// TIA Portal project "Hot Water Generation V.2 (29.01.2024)" (V15.1)

(* hardware
DEVICE "S7-1200 station_1"  S7-1200 Station
   slot 0: "Rack_0"  S7-1200 Rack  Rack  V1.0
   slot 1: "PLC_1"  CPU 1214C DC/DC/DC  6ES7 214-1AG40-0XB0  V4.2
   slot 2: "AI 4x16BIT_1"  SM 1231 AI4 x HF  6ES7 231-5ND32-0XB0  V2.0
   slot 3: "AI 4x16BIT_2"  SM 1231 AI4 x HF  6ES7 231-5ND32-0XB0  V2.0
DEVICE "HMI_1"  TP700 Comfort
   slot 0: "HMI_1"  TP700 Comfort  6AV2 124-0GC01-0AX0  15.1.0.0
   slot 1: "HMI_RT_1"  TP700 Comfort  6AV2 124-0GC01-0AX0  15.1.0.0
   slot 5: "HMI_1.IE_CP_1"  PROFINET Interface  15.0.1.0
      slot 1: "PROFINET Interface_1"  PROFINET Interface
         slot 1: "Port_1"  Port
         slot 2: "Port_2"  Port
   slot 7: "HMI_1.MPI/DP_CP_1"  MPI/DP Interface  15.0.1.0
*)

// ===== PLC "PLC_1"  CPU 1214C DC/DC/DC =====

VAR_GLOBAL   // PLC tag table "Default tag table"
   "steam_preassure_sensor_pin" AT %IW96 : Int;
   "preheating_pressure_sensor_pin" AT %IW98 : Int;
   "distribution_pressure_pin" AT %IW100 : Int;
   "preheating_temperature_input_pin" AT %IW102 : Int;
   "distribution_temperature_input_pin" AT %IW112 : Int;
   "preheating_upper_level_sensor" AT %I0.0 : Bool;
   "preheating_lower_level_sensor" AT %I0.1 : Bool;
   "distribution_upper_level_sensor" AT %I0.2 : Bool;
   "distribution_lower_level_sensor" AT %I0.3 : Bool;
   "heaters" AT %Q0.0 : Bool;
   "washing_out" AT %Q0.1 : Bool;
   "washing_in" AT %Q0.2 : Bool;
   "washing_pump" AT %Q0.3 : Bool;
   "steam_valve" AT %Q0.4 : Bool;
   "preheating_tank_comp_air_bubbling_valve" AT %Q0.5 : Bool;
   "soft_water_inlet_valve" AT %Q0.6 : Bool;
   "hot_water_transfer_valve" AT %Q0.7 : Bool;
   "distribution_tank_comp_air_bubbling_valve" AT %Q1.0 : Bool;
   "distribution_valve" AT %Q1.1 : Bool;
   "preheating_vent" AT %Q8.0 : Bool;
   "distribution_vent" AT %Q8.1 : Bool;
   "System_Byte" AT %MB1 : Byte;
   "FirstScan" AT %M1.0 : Bool;
   "DiagStatusUpdate" AT %M1.1 : Bool;
   "AlwaysTRUE" AT %M1.2 : Bool;
   "AlwaysFALSE" AT %M1.3 : Bool;
   "Clock_Byte" AT %MB0 : Byte;
   "Clock_10Hz" AT %M0.0 : Bool;
   "Clock_5Hz" AT %M0.1 : Bool;
   "Clock_2.5Hz" AT %M0.2 : Bool;
   "Clock_2Hz" AT %M0.3 : Bool;
   "Clock_1.25Hz" AT %M0.4 : Bool;
   "Clock_1Hz" AT %M0.5 : Bool;
   "Clock_0.625Hz" AT %M0.6 : Bool;
   "Clock_0.5Hz" AT %M0.7 : Bool;
   "alarm" AT %MW2 : Int;
   "steam_pressure_low" AT %M2.0 : Bool;
   "preaheating_tank_pressure_low" AT %M2.2 : Bool;
   "preaheating_tank_pressure_high" AT %M2.3 : Bool;
   "preheating_temperature_low" AT %M2.4 : Bool;
   "preheating_temperature_high" AT %M2.5 : Bool;
   "steam_pressure_high" AT %M2.1 : Bool;
   "distribution_pressure_low" AT %M2.6 : Bool;
   "distribution_pressure_high" AT %M2.7 : Bool;
   "distribution_temperature_low" AT %M3.0 : Bool;
   "distribution_temperature_high" AT %M3.1 : Bool;
   "preheating_tank_empty" AT %M3.2 : Bool;
   "distribution_tank_empty" AT %M3.3 : Bool;
   "distribution_vent_switch_inverted" AT %M4.0 : Bool;
   "preheating_tank_comp_air_bubbling_valve_switch" AT %M4.1 : Bool;
END_VAR

DATA_BLOCK "sensor_inputs"   // DB1
{ S7_Optimized_Access := 'FALSE' }
VERSION : 0.1
   VAR
      preheating_steam_preassure : Real;
      preheating_tank_pressure : Real;
      distribution_tank_pressure : Real;
      preheating_temperature : Real;
      distribution_temperature : Real;
      Trend : Struct
         DT_Max_Limit : Real;
         DT_Min_Limit : Real;
         PT_Max_Limit : Real;
         PT_Min_Limit : Real;
      END_STRUCT;
   END_VAR
BEGIN
END_DATA_BLOCK

DATA_BLOCK "setpoint"   // DB3
{ S7_Optimized_Access := 'FALSE' }
VERSION : 0.1
   VAR
      distribution_temperature : Real := 70.0;
      distribution_temperature_tolerance : Real := 2.0;
      preheating_temperature : Real := 70.0;
      preheating_temperature_tolerance : Real := 5.0;
      distribution_tank_pressure : Real := 2.5;
      preheating_tank_pressure : Real := 3.0;
      preheating_steam_pressure : Real := 3.2;
      preheating_steam_pressure_tolerance : Real := 0.5;
      preaheating_tank_pressure_tolerance : Real := 0.5;
      distribution_tank_pressure_tolerance : Real := 0.5;
      is_manual_mode : Bool;
      vent_set_pressure_during_inlet : Real := 2.5;
      vent_reset_pressure_during_inlet_off : Real := 2.0;
      vent_set_critical_pressure : Real := 3.5;
      vent_reset_critical_pressure : Real := 2.8;
      critical_temperature : Real := 85.0;
   END_VAR
BEGIN
END_DATA_BLOCK

DATA_BLOCK "state"   // DB4
{ S7_Optimized_Access := 'FALSE' }
VERSION : 0.1
   VAR
      heater_pulse : Bool;
      distribution_tank_full : Bool;
      distribution_tank_empty : Bool;
      preheating_tank_full : Bool;
      preheating_tank_empty : Bool;
      stop_distribution_controller : Bool;
      stop_preheating_controller : Bool;
      steam_pulse : Bool;
      preheating_steam_pressure_high : Bool;
      preheating_tank_pressure_high : Bool;
      emergency_stop : Bool;
      preheating_temperature_in_range : Bool;
      distribution_temperature_in_range : Bool;
   END_VAR
BEGIN
END_DATA_BLOCK

DATA_BLOCK "read_sensors_DB"   // DB6
{ S7_Optimized_Access := 'TRUE' }
VERSION : 0.1
// stored: InstanceOfName read_sensors
"read_sensors"
BEGIN
END_DATA_BLOCK

DATA_BLOCK "manual"   // DB7
{ S7_Optimized_Access := 'FALSE' }
VERSION : 0.1
   VAR
      steam_valve : Bool;
      preheating_tank_comp_air_valve : Bool;
      soft_water_inlet_valve : Bool;
      hot_water_transfer_valve : Bool;
      distribution_tank_comp_air_valve : Bool;
      distribution_valve : Bool;
      heater : Bool;
      preheating_vent : Bool;
      distribution_vent : Bool;
   END_VAR
BEGIN
END_DATA_BLOCK

DATA_BLOCK "control_valves"   // DB8
{ S7_Optimized_Access := 'TRUE' }
VERSION : 0.1
// stored: InstanceOfName control_valve
"control_valve"
BEGIN
END_DATA_BLOCK

DATA_BLOCK "alarm_limit"   // DB9
{ S7_Optimized_Access := 'FALSE' }
VERSION : 0.1
   VAR
      steam_pressure_low : Real;
      steam_pressure_low_delay : Time;
      steam_pressure_high : Real;
      steam_pressure_high_delay : Time;
      preaheating_tank_pressure_low : Real;
      preaheating_tank_pressure_low_delay : Time;
      preaheating_tank_pressure_high : Real;
      preaheating_tank_pressure_high_delay : Time;
      preheating_temperature_low : Real;
      preheating_temperature_low_delay : Time;
      preheating_temperature_high : Real;
      preheating_temperature_high_delay : Time;
      distribution_pressure_low : Real;
      distribution_pressure_low_delay : Time;
      distribution_pressure_high : Real;
      distribution_pressure_high_delay : Time;
      distribution_temperature_low : Real;
      distribution_temperature_low_delay : Time;
      distribution_temperature_high : Real;
      distribution_temperature_high_delay : Time;
      preheating_tank_empty : Real;
      preheating_tank_empty_delay : Time;
      distribution_tank_empty : Real;
      distribution_tank_empty_delay : Time;
   END_VAR
BEGIN
END_DATA_BLOCK

DATA_BLOCK "alarm_management_DB"   // DB10
{ S7_Optimized_Access := 'TRUE' }
VERSION : 0.1
// stored: InstanceOfName alarm_management
"alarm_management"
BEGIN
END_DATA_BLOCK

FUNCTION_BLOCK "analog_input"   // FB1, LAD
{ S7_Optimized_Access := 'TRUE' }
VERSION : 0.1
   VAR_INPUT
      sensor_min : Real;
      sensor_max : Real;
      sensor_address : Int;
   END_VAR
   VAR_OUTPUT
      Calibrated_value : Real;
   END_VAR
   VAR
      Calibration : Real;
      Scaled_value : Real;
   END_VAR
   VAR_TEMP
      norm : Real;
   END_VAR
BEGIN

REGION Network 1
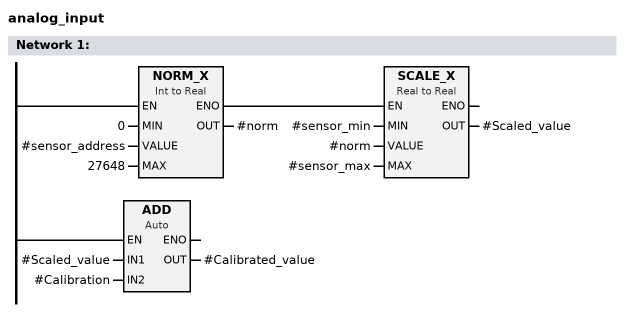
   RUNG wire#powerrail
      { S7_Templates := "[SrcType := Int, DestType := Real]" } Normalize(min := 0, value := #sensor_address, max := 27648, out => #norm)
      { S7_Templates := "[SrcType := Real, DestType := Real]" } Scale(min := #sensor_min, value := #norm, max := #sensor_max, out => #Scaled_value)
   END_RUNG
   RUNG wire#powerrail
      Add(in1 := #Scaled_value, in2 := #Calibration, out => #Calibrated_value)
   END_RUNG
   // the same network as SCL:
   #norm := NORM_X(MIN := 0, VALUE := #sensor_address, MAX := 27648);
   #Scaled_value := SCALE_X(MIN := #sensor_min, VALUE := #norm, MAX := #sensor_max);
   #Calibrated_value := #Scaled_value + #Calibration;
END_REGION
END_FUNCTION_BLOCK

FUNCTION_BLOCK "read_sensors"   // FB2, LAD
{ S7_Optimized_Access := 'TRUE' }
VERSION : 0.1
   VAR
      Steam_pressure_input : "analog_input";
      preheating_tank_pressure_input : "analog_input";
      distribution_tank_pressure_input : "analog_input";
      preheating_temperature_input : "analog_input";
      distribution_temperature_input : "analog_input";
   END_VAR
BEGIN

REGION Network 1
   // Pressure sensors
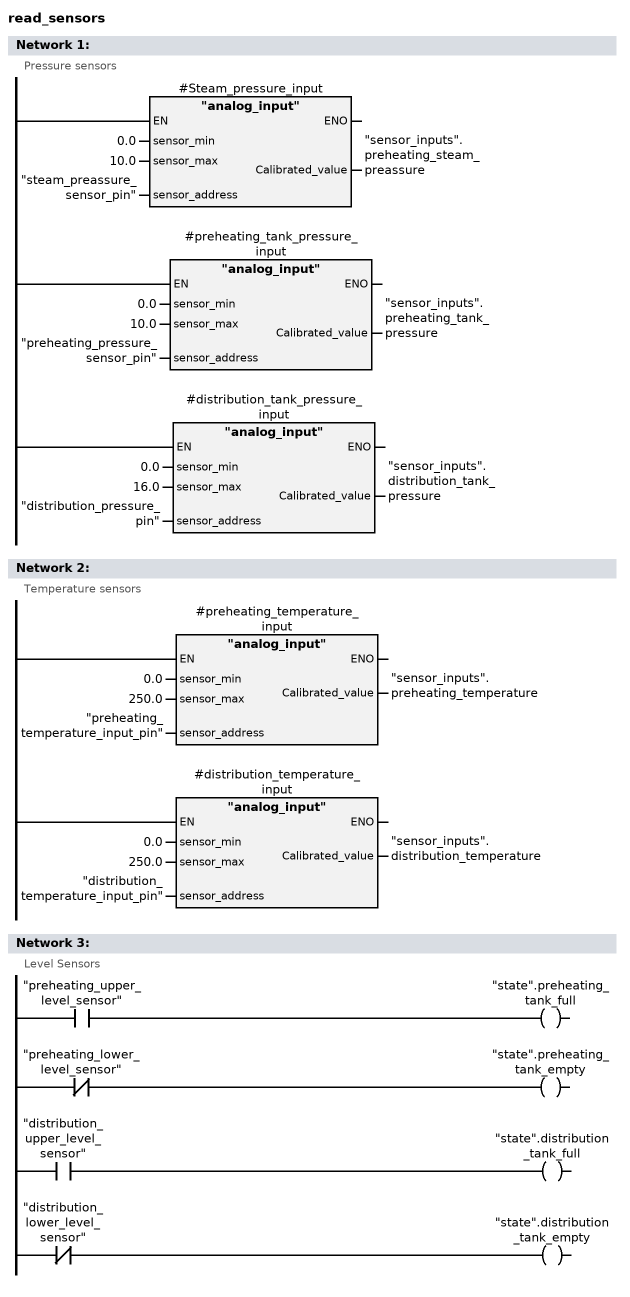
   RUNG wire#powerrail
      #Steam_pressure_input(sensor_min := 0.0, sensor_max := 10.0, sensor_address := "steam_preassure_sensor_pin", Calibrated_value => "sensor_inputs".preheating_steam_preassure)
   END_RUNG
   RUNG wire#powerrail
      #preheating_tank_pressure_input(sensor_min := 0.0, sensor_max := 10.0, sensor_address := "preheating_pressure_sensor_pin", Calibrated_value => "sensor_inputs".preheating_tank_pressure)
   END_RUNG
   RUNG wire#powerrail
      #distribution_tank_pressure_input(sensor_min := 0.0, sensor_max := 16.0, sensor_address := "distribution_pressure_pin", Calibrated_value => "sensor_inputs".distribution_tank_pressure)
   END_RUNG
   // the same network as SCL:
   #Steam_pressure_input(sensor_min := 0.0,   // "analog_input"
                         sensor_max := 10.0,
                         sensor_address := "steam_preassure_sensor_pin",
                         Calibrated_value => "sensor_inputs".preheating_steam_preassure);
   #preheating_tank_pressure_input(sensor_min := 0.0,   // "analog_input"
                           sensor_max := 10.0,
                           sensor_address := "preheating_pressure_sensor_pin",
                           Calibrated_value => "sensor_inputs".preheating_tank_pressure);
   #distribution_tank_pressure_input(sensor_min := 0.0,   // "analog_input"
                           sensor_max := 16.0,
                           sensor_address := "distribution_pressure_pin",
                           Calibrated_value => "sensor_inputs".distribution_tank_pressure);
END_REGION

REGION Network 2
   // Temperature sensors
   RUNG wire#powerrail
      #preheating_temperature_input(sensor_min := 0.0, sensor_max := 250.0, sensor_address := "preheating_temperature_input_pin", Calibrated_value => "sensor_inputs".preheating_temperature)
   END_RUNG
   RUNG wire#powerrail
      #distribution_temperature_input(sensor_min := 0.0, sensor_max := 250.0, sensor_address := "distribution_temperature_input_pin", Calibrated_value => "sensor_inputs".distribution_temperature)
   END_RUNG
   // the same network as SCL:
   #preheating_temperature_input(sensor_min := 0.0,   // "analog_input"
                           sensor_max := 250.0,
                           sensor_address := "preheating_temperature_input_pin",
                           Calibrated_value => "sensor_inputs".preheating_temperature);
   #distribution_temperature_input(sensor_min := 0.0,   // "analog_input"
                           sensor_max := 250.0,
                           sensor_address := "distribution_temperature_input_pin",
                           Calibrated_value => "sensor_inputs".distribution_temperature);
END_REGION

REGION Network 3
   // Level Sensors
   RUNG wire#powerrail
      Contact( "preheating_upper_level_sensor" )
      Coil( "state".preheating_tank_full )
   END_RUNG
   RUNG wire#powerrail
      I_Contact( "preheating_lower_level_sensor" )
      Coil( "state".preheating_tank_empty )
   END_RUNG
   RUNG wire#powerrail
      Contact( "distribution_upper_level_sensor" )
      Coil( "state".distribution_tank_full )
   END_RUNG
   RUNG wire#powerrail
      I_Contact( "distribution_lower_level_sensor" )
      Coil( "state".distribution_tank_empty )
   END_RUNG
   // the same network as SCL:
   "state".preheating_tank_full := "preheating_upper_level_sensor";
   "state".preheating_tank_empty := NOT "preheating_lower_level_sensor";
   "state".distribution_tank_full := "distribution_upper_level_sensor";
   "state".distribution_tank_empty := NOT "distribution_lower_level_sensor";
END_REGION
END_FUNCTION_BLOCK

FUNCTION_BLOCK "valve_controller_within_range"   // FB3, LAD
{ S7_Optimized_Access := 'TRUE' }
VERSION : 0.1
   VAR_INPUT
      setpoint : Real;
      current : Real;
      tolerance : Real;
      manual_switch : Bool;
   END_VAR
   VAR_OUTPUT
      output : Bool;
   END_VAR
   VAR_TEMP
      lower_trigger_point : Real;
      higher_trigger_point : Real;
   END_VAR
BEGIN

REGION Network 1
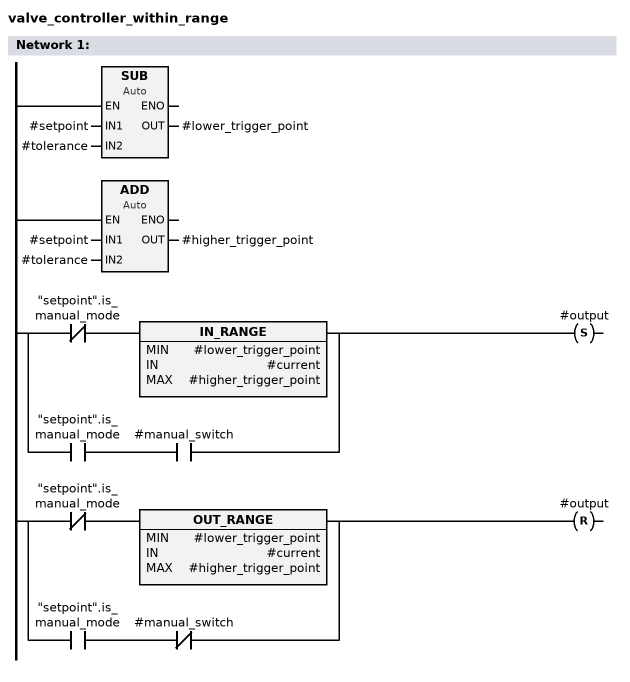
   #lower_trigger_point := #setpoint - #tolerance;
   #higher_trigger_point := #setpoint + #tolerance;
   IF (NOT "setpoint".is_manual_mode AND (#lower_trigger_point <= #current) AND (#current <= #higher_trigger_point)) OR ("setpoint".is_manual_mode AND #manual_switch) THEN
       #output := TRUE;
   END_IF;
   IF (NOT "setpoint".is_manual_mode AND ((#current < #lower_trigger_point) OR (#current > #higher_trigger_point))) OR ("setpoint".is_manual_mode AND NOT #manual_switch) THEN
       #output := FALSE;
   END_IF;
END_REGION
END_FUNCTION_BLOCK

FUNCTION_BLOCK "pressure_controller"   // FB4, LAD
{ S7_Optimized_Access := 'TRUE' }
VERSION : 0.1
   VAR
      tank_1_steam_valve_controller : "valve_controller_within_range";
   END_VAR
BEGIN

REGION Network 1
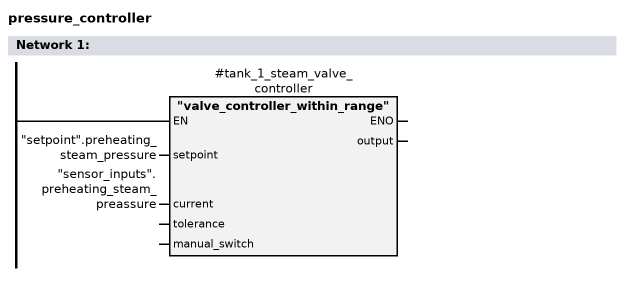
   RUNG wire#powerrail
      #tank_1_steam_valve_controller(setpoint := "setpoint".preheating_steam_pressure, current := "sensor_inputs".preheating_steam_preassure, tolerance :=, output =>, manual_switch :=)
   END_RUNG
   // the same network as SCL:
   #tank_1_steam_valve_controller(setpoint := "setpoint".preheating_steam_pressure,   // "valve_controller_within_range"
                           current := "sensor_inputs".preheating_steam_preassure);
END_REGION
END_FUNCTION_BLOCK

FUNCTION_BLOCK "control_valve"   // FB5, LAD
{ S7_Optimized_Access := 'TRUE' }
VERSION : 0.1
   VAR
      distribution_tank_fillup_timer : TON_TIME;
      hot_water_transfer_valve_controller : "valve_controller_within_range";
      distribution_valve_timer : TON_TIME;
      preheating_pressure_valve_controller : "valve_controller_bellow_high_limit";
      distribution_pressure_valve_controller : "valve_controller_bellow_high_limit";
      distribution_valve_controller : "valve_controller_within_range";
      vent_valve_controller_within_range_DB : "valve_controller_within_range";
      distribution_vent_valve_controller_bellow_high_limit_DB : "valve_controller_bellow_high_limit";
   END_VAR
   VAR_TEMP   // added for the SCL form of the ladder/FBD networks
      _w1 : Bool;
      _w2 : Bool;
   END_VAR
BEGIN

REGION Network 1: Preheating tank pressure
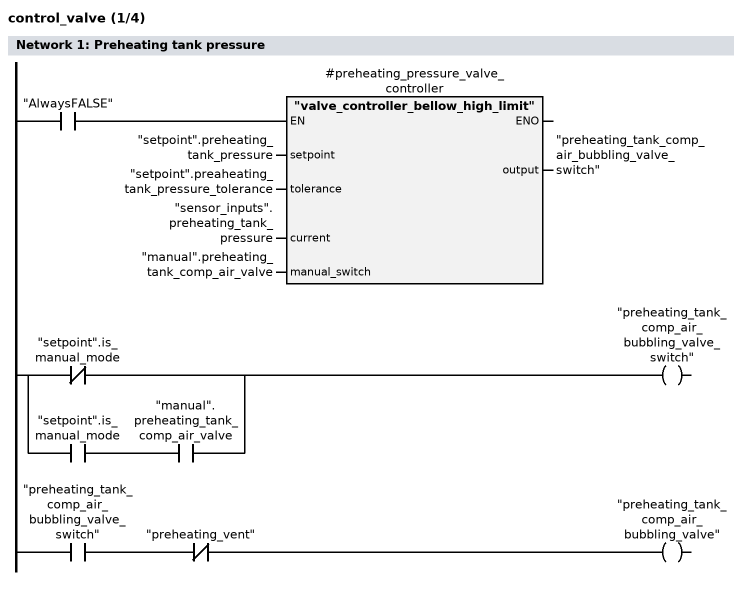
   RUNG wire#powerrail
      Contact( "AlwaysFALSE" )
      #preheating_pressure_valve_controller(setpoint := "setpoint".preheating_tank_pressure, tolerance := "setpoint".preaheating_tank_pressure_tolerance, current := "sensor_inputs".preheating_tank_pressure, manual_switch := "manual".preheating_tank_comp_air_valve, output => "preheating_tank_comp_air_bubbling_valve_switch")
   END_RUNG
   RUNG wire#powerrail
      I_Contact( "setpoint".is_manual_mode )
      wire#w1
      Coil( "preheating_tank_comp_air_bubbling_valve_switch" )
   END_RUNG
   RUNG wire#powerrail
      Contact( "setpoint".is_manual_mode )
      Contact( "manual".preheating_tank_comp_air_valve )
   END_RUNG wire#w1
   RUNG wire#powerrail
      Contact( "preheating_tank_comp_air_bubbling_valve_switch" )
      I_Contact( "preheating_vent" )
      Coil( "preheating_tank_comp_air_bubbling_valve" )
   END_RUNG
   // the same network as SCL:
   IF "AlwaysFALSE" THEN
       #preheating_pressure_valve_controller(setpoint := "setpoint".preheating_tank_pressure,   // "valve_controller_bellow_high_limit"
                               tolerance := "setpoint".preaheating_tank_pressure_tolerance,
                               current := "sensor_inputs".preheating_tank_pressure,
                               manual_switch := "manual".preheating_tank_comp_air_valve,
                               output => "preheating_tank_comp_air_bubbling_valve_switch");
   END_IF;
   "preheating_tank_comp_air_bubbling_valve_switch" := NOT "setpoint".is_manual_mode OR ("setpoint".is_manual_mode AND "manual".preheating_tank_comp_air_valve);
   "preheating_tank_comp_air_bubbling_valve" := "preheating_tank_comp_air_bubbling_valve_switch" AND NOT "preheating_vent";
END_REGION

REGION Network 2: Preheating inlet water
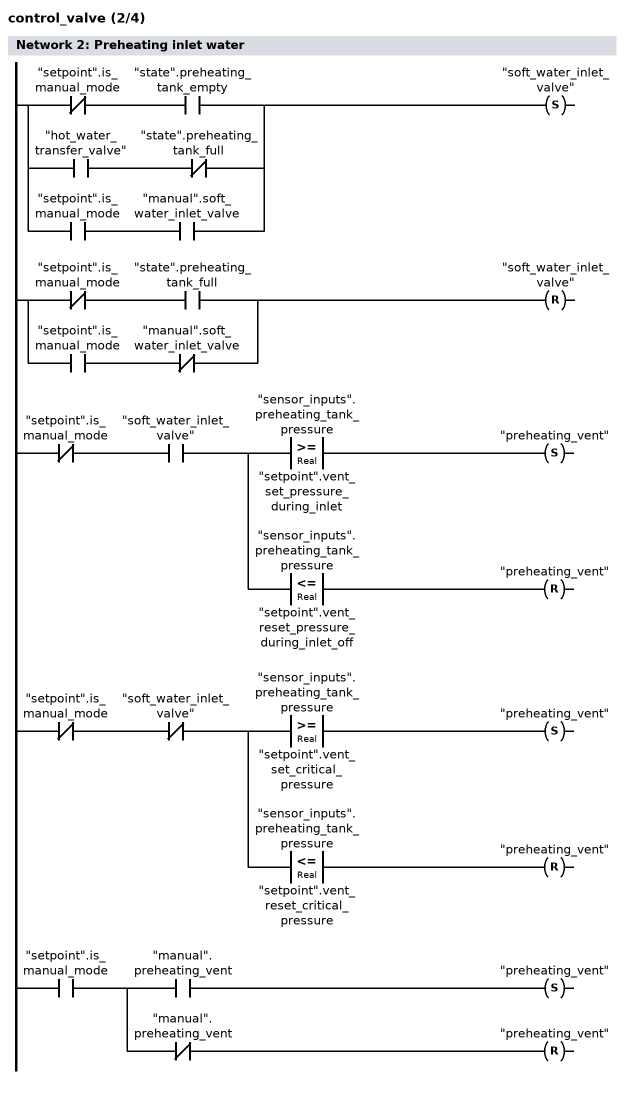
   RUNG wire#powerrail
      I_Contact( "setpoint".is_manual_mode )
      Contact( "state".preheating_tank_empty )
      wire#w1
      S_Coil( "soft_water_inlet_valve" )
   END_RUNG
   RUNG wire#powerrail
      Contact( "hot_water_transfer_valve" )
      I_Contact( "state".preheating_tank_full )
   END_RUNG wire#w1
   RUNG wire#powerrail
      Contact( "setpoint".is_manual_mode )
      Contact( "manual".soft_water_inlet_valve )
   END_RUNG wire#w1
   RUNG wire#powerrail
      I_Contact( "setpoint".is_manual_mode )
      Contact( "state".preheating_tank_full )
      wire#w2
      R_Coil( "soft_water_inlet_valve" )
   END_RUNG
   RUNG wire#powerrail
      Contact( "setpoint".is_manual_mode )
      I_Contact( "manual".soft_water_inlet_valve )
   END_RUNG wire#w2
   RUNG wire#powerrail
      I_Contact( "setpoint".is_manual_mode )
      Contact( "soft_water_inlet_valve" )
      wire#w3
      { S7_Templates := "SrcType := Real" } GE_Contact(in1 := "sensor_inputs".preheating_tank_pressure, in2 := "setpoint".vent_set_pressure_during_inlet)
      S_Coil( "preheating_vent" )
   END_RUNG
   RUNG wire#w3
      { S7_Templates := "SrcType := Real" } LE_Contact(in1 := "sensor_inputs".preheating_tank_pressure, in2 := "setpoint".vent_reset_pressure_during_inlet_off)
      R_Coil( "preheating_vent" )
   END_RUNG
   RUNG wire#powerrail
      I_Contact( "setpoint".is_manual_mode )
      I_Contact( "soft_water_inlet_valve" )
      wire#w4
      { S7_Templates := "SrcType := Real" } GE_Contact(in1 := "sensor_inputs".preheating_tank_pressure, in2 := "setpoint".vent_set_critical_pressure)
      S_Coil( "preheating_vent" )
   END_RUNG
   RUNG wire#w4
      { S7_Templates := "SrcType := Real" } LE_Contact(in1 := "sensor_inputs".preheating_tank_pressure, in2 := "setpoint".vent_reset_critical_pressure)
      R_Coil( "preheating_vent" )
   END_RUNG
   RUNG wire#powerrail
      Contact( "setpoint".is_manual_mode )
      wire#w5
      Contact( "manual".preheating_vent )
      S_Coil( "preheating_vent" )
   END_RUNG
   RUNG wire#w5
      I_Contact( "manual".preheating_vent )
      R_Coil( "preheating_vent" )
   END_RUNG
   // the same network as SCL:
   IF (NOT "setpoint".is_manual_mode AND "state".preheating_tank_empty) OR ("hot_water_transfer_valve" AND NOT "state".preheating_tank_full) OR ("setpoint".is_manual_mode AND "manual".soft_water_inlet_valve) THEN
       "soft_water_inlet_valve" := TRUE;
   END_IF;
   IF (NOT "setpoint".is_manual_mode AND "state".preheating_tank_full) OR ("setpoint".is_manual_mode AND NOT "manual".soft_water_inlet_valve) THEN
       "soft_water_inlet_valve" := FALSE;
   END_IF;
   #_w1 := NOT "setpoint".is_manual_mode AND "soft_water_inlet_valve";
   IF #_w1 AND ("sensor_inputs".preheating_tank_pressure >= "setpoint".vent_set_pressure_during_inlet) THEN
       "preheating_vent" := TRUE;
   END_IF;
   IF #_w1 AND ("sensor_inputs".preheating_tank_pressure <= "setpoint".vent_reset_pressure_during_inlet_off) THEN
       "preheating_vent" := FALSE;
   END_IF;
   #_w2 := NOT "setpoint".is_manual_mode AND NOT "soft_water_inlet_valve";
   IF #_w2 AND ("sensor_inputs".preheating_tank_pressure >= "setpoint".vent_set_critical_pressure) THEN
       "preheating_vent" := TRUE;
   END_IF;
   IF #_w2 AND ("sensor_inputs".preheating_tank_pressure <= "setpoint".vent_reset_critical_pressure) THEN
       "preheating_vent" := FALSE;
   END_IF;
   IF "setpoint".is_manual_mode AND "manual".preheating_vent THEN "preheating_vent" := TRUE; END_IF;
   IF "setpoint".is_manual_mode AND NOT "manual".preheating_vent THEN "preheating_vent" := FALSE; END_IF;
END_REGION

REGION Network 3: Preheated water transfer
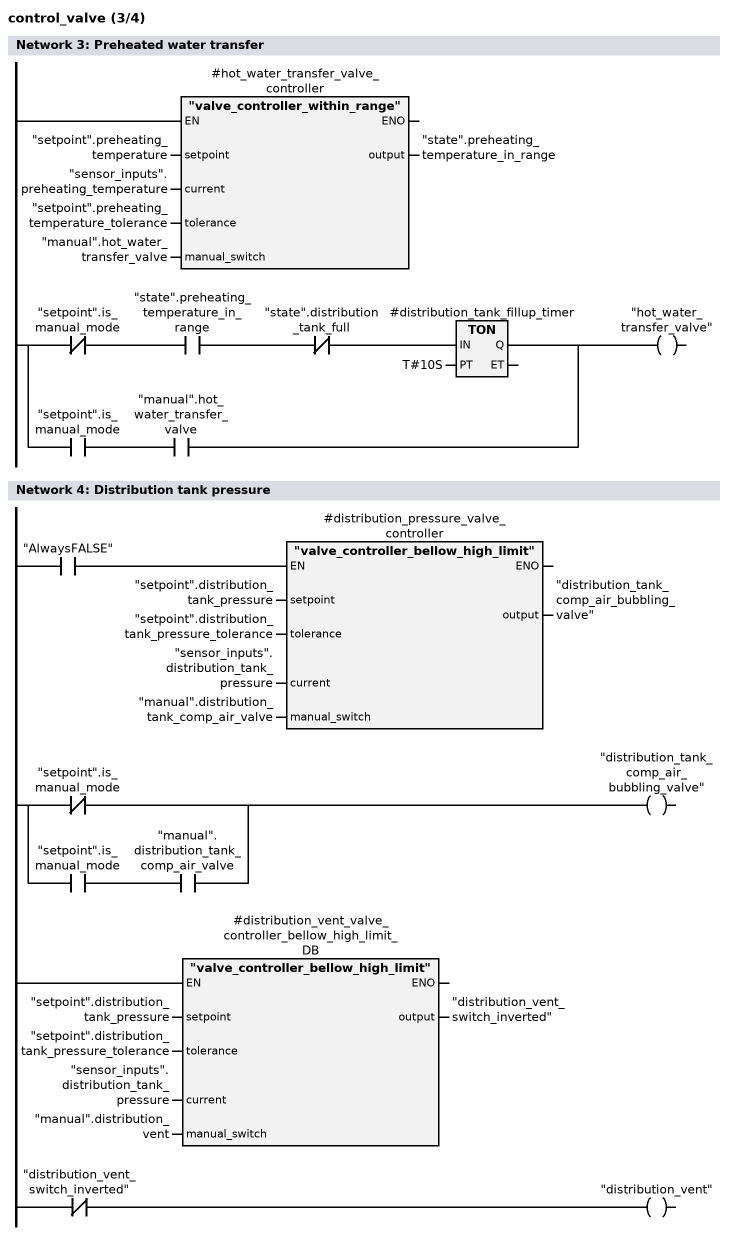
   #hot_water_transfer_valve_controller(setpoint := "setpoint".preheating_temperature,   // "valve_controller_within_range"
                           current := "sensor_inputs".preheating_temperature,
                           tolerance := "setpoint".preheating_temperature_tolerance,
                           manual_switch := "manual".hot_water_transfer_valve,
                           output => "state".preheating_temperature_in_range);
   #distribution_tank_fillup_timer(IN := NOT "setpoint".is_manual_mode AND "state".preheating_temperature_in_range AND NOT "state".distribution_tank_full,   // TON
                           PT := T#10S);
   "hot_water_transfer_valve" := #distribution_tank_fillup_timer.Q OR ("setpoint".is_manual_mode AND "manual".hot_water_transfer_valve);
END_REGION

REGION Network 4: Distribution tank pressure
   RUNG wire#powerrail
      Contact( "AlwaysFALSE" )
      #distribution_pressure_valve_controller(setpoint := "setpoint".distribution_tank_pressure, tolerance := "setpoint".distribution_tank_pressure_tolerance, current := "sensor_inputs".distribution_tank_pressure, manual_switch := "manual".distribution_tank_comp_air_valve, output => "distribution_tank_comp_air_bubbling_valve")
   END_RUNG
   RUNG wire#powerrail
      I_Contact( "setpoint".is_manual_mode )
      wire#w1
      Coil( "distribution_tank_comp_air_bubbling_valve" )
   END_RUNG
   RUNG wire#powerrail
      Contact( "setpoint".is_manual_mode )
      Contact( "manual".distribution_tank_comp_air_valve )
   END_RUNG wire#w1
   RUNG wire#powerrail
      #distribution_vent_valve_controller_bellow_high_limit_DB(setpoint := "setpoint".distribution_tank_pressure, tolerance := "setpoint".distribution_tank_pressure_tolerance, current := "sensor_inputs".distribution_tank_pressure, manual_switch := "manual".distribution_vent, output => "distribution_vent_switch_inverted")
   END_RUNG
   RUNG wire#powerrail
      I_Contact( "distribution_vent_switch_inverted" )
      Coil( "distribution_vent" )
   END_RUNG
   // the same network as SCL:
   IF "AlwaysFALSE" THEN
       #distribution_pressure_valve_controller(setpoint := "setpoint".distribution_tank_pressure,   // "valve_controller_bellow_high_limit"
                               tolerance := "setpoint".distribution_tank_pressure_tolerance,
                               current := "sensor_inputs".distribution_tank_pressure,
                               manual_switch := "manual".distribution_tank_comp_air_valve,
                               output => "distribution_tank_comp_air_bubbling_valve");
   END_IF;
   "distribution_tank_comp_air_bubbling_valve" := NOT "setpoint".is_manual_mode OR ("setpoint".is_manual_mode AND "manual".distribution_tank_comp_air_valve);
   #distribution_vent_valve_controller_bellow_high_limit_DB(setpoint := "setpoint".distribution_tank_pressure,   // "valve_controller_bellow_high_limit"
                           tolerance := "setpoint".distribution_tank_pressure_tolerance,
                           current := "sensor_inputs".distribution_tank_pressure,
                           manual_switch := "manual".distribution_vent,
                           output => "distribution_vent_switch_inverted");
   "distribution_vent" := NOT "distribution_vent_switch_inverted";
END_REGION

REGION Network 5: Ditribution control
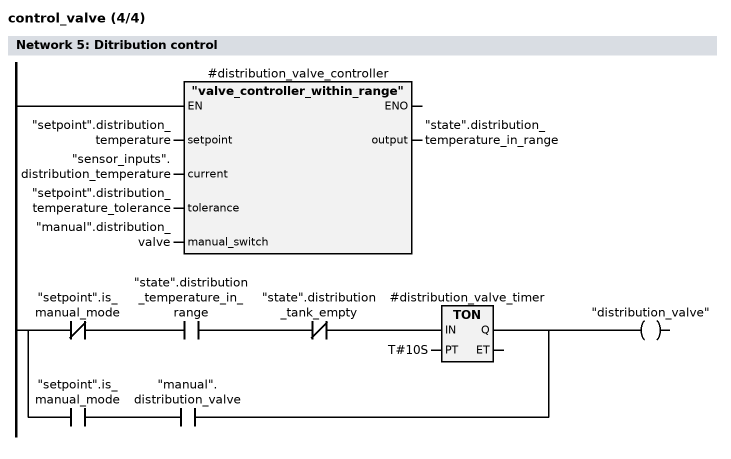
   #distribution_valve_controller(setpoint := "setpoint".distribution_temperature,   // "valve_controller_within_range"
                           current := "sensor_inputs".distribution_temperature,
                           tolerance := "setpoint".distribution_temperature_tolerance,
                           manual_switch := "manual".distribution_valve,
                           output => "state".distribution_temperature_in_range);
   #distribution_valve_timer(IN := NOT "setpoint".is_manual_mode AND "state".distribution_temperature_in_range AND NOT "state".distribution_tank_empty,   // TON
                           PT := T#10S);
   "distribution_valve" := #distribution_valve_timer.Q OR ("setpoint".is_manual_mode AND "manual".distribution_valve);
END_REGION
END_FUNCTION_BLOCK

FUNCTION_BLOCK "valve_controller_bellow_high_limit"   // FB6, LAD
{ S7_Optimized_Access := 'TRUE' }
VERSION : 0.1
   VAR_INPUT
      setpoint : Real;
      tolerance : Real;
      current : Real;
      manual_switch : Bool;
   END_VAR
   VAR_OUTPUT
      output : Bool;
   END_VAR
   VAR_TEMP
      lower_trigger_point : Real;
   END_VAR
BEGIN

REGION Network 1
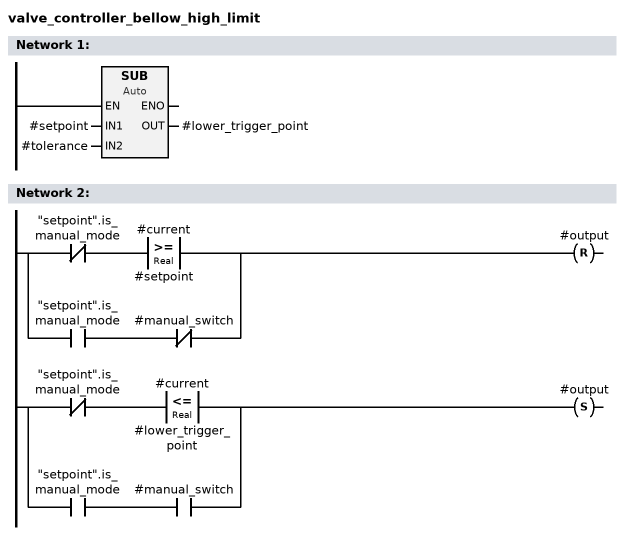
   RUNG wire#powerrail
      Sub(in1 := #setpoint, in2 := #tolerance, out => #lower_trigger_point)
   END_RUNG
   // the same network as SCL:
   #lower_trigger_point := #setpoint - #tolerance;
END_REGION

REGION Network 2
   RUNG wire#powerrail
      I_Contact( "setpoint".is_manual_mode )
      { S7_Templates := "SrcType := Real" } GE_Contact(in1 := #current, in2 := #setpoint)
      wire#w1
      R_Coil( #output )
   END_RUNG
   RUNG wire#powerrail
      Contact( "setpoint".is_manual_mode )
      I_Contact( #manual_switch )
   END_RUNG wire#w1
   RUNG wire#powerrail
      I_Contact( "setpoint".is_manual_mode )
      { S7_Templates := "SrcType := Real" } LE_Contact(in1 := #current, in2 := #lower_trigger_point)
      wire#w2
      S_Coil( #output )
   END_RUNG
   RUNG wire#powerrail
      Contact( "setpoint".is_manual_mode )
      Contact( #manual_switch )
   END_RUNG wire#w2
   // the same network as SCL:
   IF (NOT "setpoint".is_manual_mode AND (#current >= #setpoint)) OR ("setpoint".is_manual_mode AND NOT #manual_switch) THEN
       #output := FALSE;
   END_IF;
   IF (NOT "setpoint".is_manual_mode AND (#current <= #lower_trigger_point)) OR ("setpoint".is_manual_mode AND #manual_switch) THEN
       #output := TRUE;
   END_IF;
END_REGION
END_FUNCTION_BLOCK

FUNCTION_BLOCK "alarm_management"   // FB7, LAD
{ S7_Optimized_Access := 'TRUE' }
VERSION : 0.1
   VAR
      steam_pressure_low_delay_timer : TON_TIME;
      steam_pressure_low_high_timer : TON_TIME;
      prehearting_tank_pressure_low_timer : TON_TIME;
      prehearting_tank_pressure_high_timer : TON_TIME;
      preheating_temperature_low_timer : TON_TIME;
      preheating_temperature_high_timer : TON_TIME;
      distribution_tank_pressure_high_timer : TON_TIME;
      distribution_tank_pressure_low_timer : TON_TIME;
      distribution_temperature_low_timer : TON_TIME;
      distribution_temperature_high_timer : TON_TIME;
      preheating_tank_empty_timer : TON_TIME;
      distribution_tank_empty_timer : TON_TIME;
   END_VAR
BEGIN

REGION Network 1
   // Preheating
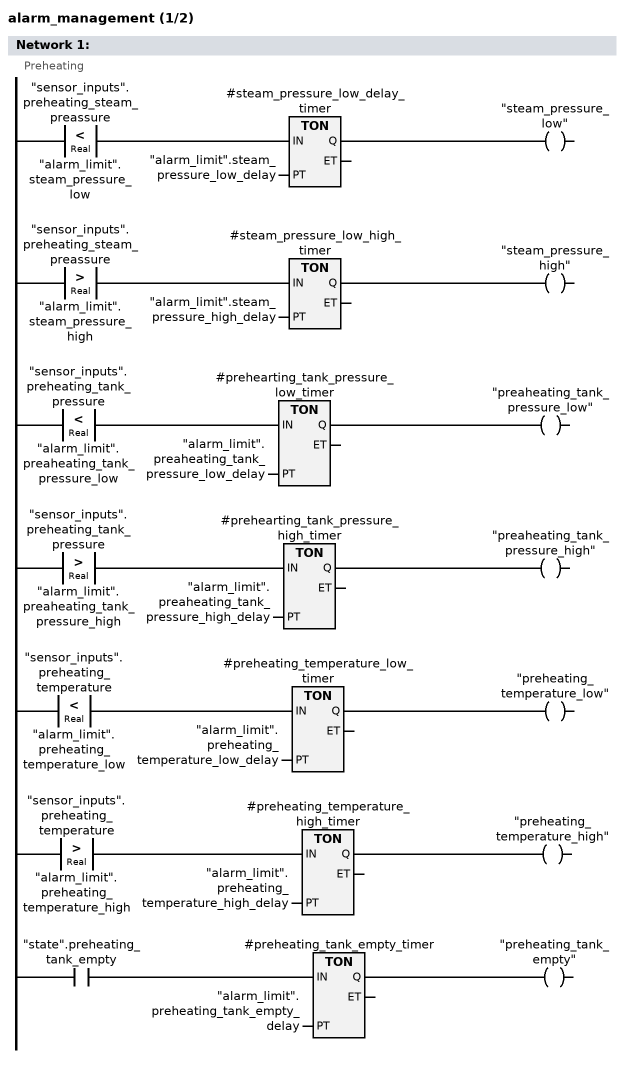
   #steam_pressure_low_delay_timer(IN := "sensor_inputs".preheating_steam_preassure < "alarm_limit".steam_pressure_low,   // TON
                           PT := "alarm_limit".steam_pressure_low_delay);
   "steam_pressure_low" := #steam_pressure_low_delay_timer.Q;
   #steam_pressure_low_high_timer(IN := "sensor_inputs".preheating_steam_preassure > "alarm_limit".steam_pressure_high,   // TON
                           PT := "alarm_limit".steam_pressure_high_delay);
   "steam_pressure_high" := #steam_pressure_low_high_timer.Q;
   #prehearting_tank_pressure_low_timer(IN := "sensor_inputs".preheating_tank_pressure < "alarm_limit".preaheating_tank_pressure_low,   // TON
                           PT := "alarm_limit".preaheating_tank_pressure_low_delay);
   "preaheating_tank_pressure_low" := #prehearting_tank_pressure_low_timer.Q;
   #prehearting_tank_pressure_high_timer(IN := "sensor_inputs".preheating_tank_pressure > "alarm_limit".preaheating_tank_pressure_high,   // TON
                           PT := "alarm_limit".preaheating_tank_pressure_high_delay);
   "preaheating_tank_pressure_high" := #prehearting_tank_pressure_high_timer.Q;
   #preheating_temperature_low_timer(IN := "sensor_inputs".preheating_temperature < "alarm_limit".preheating_temperature_low,   // TON
                           PT := "alarm_limit".preheating_temperature_low_delay);
   "preheating_temperature_low" := #preheating_temperature_low_timer.Q;
   #preheating_temperature_high_timer(IN := "sensor_inputs".preheating_temperature > "alarm_limit".preheating_temperature_high,   // TON
                           PT := "alarm_limit".preheating_temperature_high_delay);
   "preheating_temperature_high" := #preheating_temperature_high_timer.Q;
   #preheating_tank_empty_timer(IN := "state".preheating_tank_empty,   // TON
                           PT := "alarm_limit".preheating_tank_empty_delay);
   "preheating_tank_empty" := #preheating_tank_empty_timer.Q;
END_REGION

REGION Network 2
   // Distribution
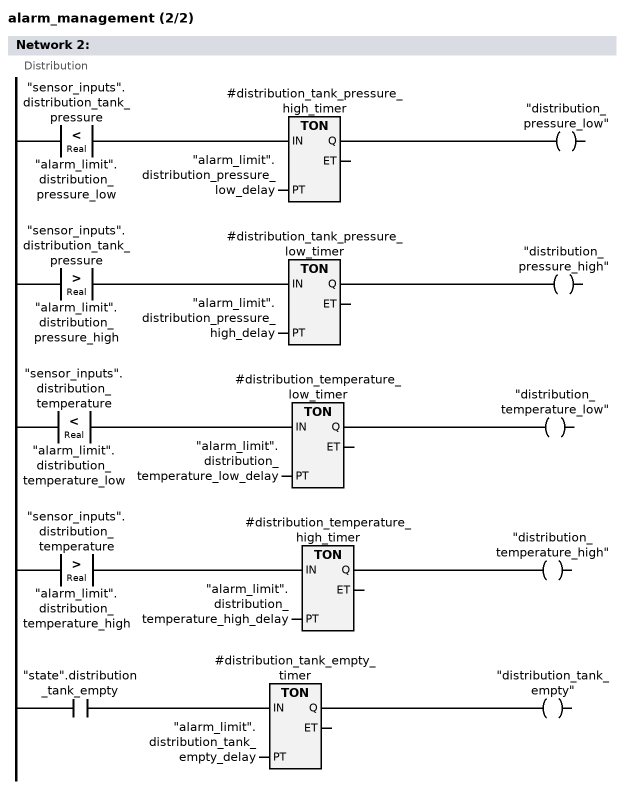
   #distribution_tank_pressure_high_timer(IN := "sensor_inputs".distribution_tank_pressure < "alarm_limit".distribution_pressure_low,   // TON
                           PT := "alarm_limit".distribution_pressure_low_delay);
   "distribution_pressure_low" := #distribution_tank_pressure_high_timer.Q;
   #distribution_tank_pressure_low_timer(IN := "sensor_inputs".distribution_tank_pressure > "alarm_limit".distribution_pressure_high,   // TON
                           PT := "alarm_limit".distribution_pressure_high_delay);
   "distribution_pressure_high" := #distribution_tank_pressure_low_timer.Q;
   #distribution_temperature_low_timer(IN := "sensor_inputs".distribution_temperature < "alarm_limit".distribution_temperature_low,   // TON
                           PT := "alarm_limit".distribution_temperature_low_delay);
   "distribution_temperature_low" := #distribution_temperature_low_timer.Q;
   #distribution_temperature_high_timer(IN := "sensor_inputs".distribution_temperature > "alarm_limit".distribution_temperature_high,   // TON
                           PT := "alarm_limit".distribution_temperature_high_delay);
   "distribution_temperature_high" := #distribution_temperature_high_timer.Q;
   #distribution_tank_empty_timer(IN := "state".distribution_tank_empty,   // TON
                           PT := "alarm_limit".distribution_tank_empty_delay);
   "distribution_tank_empty" := #distribution_tank_empty_timer.Q;
END_REGION
END_FUNCTION_BLOCK

FUNCTION_BLOCK "descaling"   // FB8, LAD
{ S7_Optimized_Access := 'TRUE' }
VERSION : 0.1
BEGIN
END_FUNCTION_BLOCK

FUNCTION_BLOCK "valve_controller_above_low_limit"   // FB9, LAD
{ S7_Optimized_Access := 'TRUE' }
VERSION : 0.1
   VAR_INPUT
      setpoint : Real;
      tolerance : Real;
      current : Real;
      manual_switch : Bool;
   END_VAR
   VAR_OUTPUT
      output : Bool;
   END_VAR
   VAR_TEMP
      higher_trigger_point : Real;
   END_VAR
BEGIN

REGION Network 1
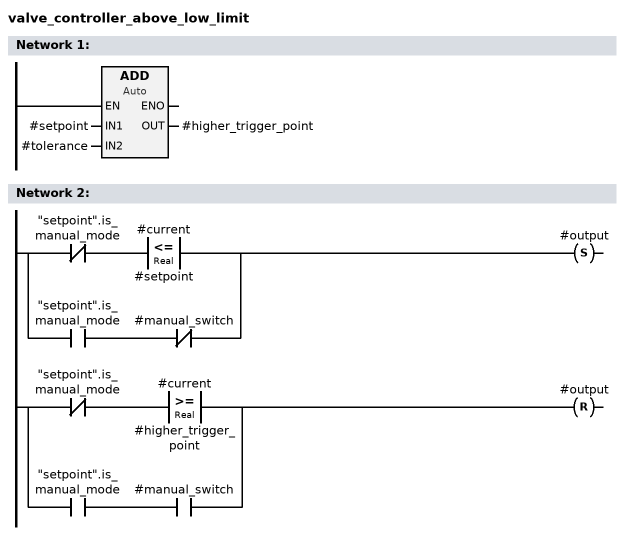
   RUNG wire#powerrail
      Add(in1 := #setpoint, in2 := #tolerance, out => #higher_trigger_point)
   END_RUNG
   // the same network as SCL:
   #higher_trigger_point := #setpoint + #tolerance;
END_REGION

REGION Network 2
   RUNG wire#powerrail
      I_Contact( "setpoint".is_manual_mode )
      { S7_Templates := "SrcType := Real" } LE_Contact(in1 := #current, in2 := #setpoint)
      wire#w1
      S_Coil( #output )
   END_RUNG
   RUNG wire#powerrail
      Contact( "setpoint".is_manual_mode )
      I_Contact( #manual_switch )
   END_RUNG wire#w1
   RUNG wire#powerrail
      I_Contact( "setpoint".is_manual_mode )
      { S7_Templates := "SrcType := Real" } GE_Contact(in1 := #current, in2 := #higher_trigger_point)
      wire#w2
      R_Coil( #output )
   END_RUNG
   RUNG wire#powerrail
      Contact( "setpoint".is_manual_mode )
      Contact( #manual_switch )
   END_RUNG wire#w2
   // the same network as SCL:
   IF (NOT "setpoint".is_manual_mode AND (#current <= #setpoint)) OR ("setpoint".is_manual_mode AND NOT #manual_switch) THEN
       #output := TRUE;
   END_IF;
   IF (NOT "setpoint".is_manual_mode AND (#current >= #higher_trigger_point)) OR ("setpoint".is_manual_mode AND #manual_switch) THEN
       #output := FALSE;
   END_IF;
END_REGION
END_FUNCTION_BLOCK

ORGANIZATION_BLOCK "Main"   // OB1, LAD, ProgramCycle
TITLE = "Main Program Sweep (Cycle)"
{ S7_Optimized_Access := 'TRUE' }
VERSION : 0.1
   VAR_INPUT
      Initial_Call : Bool;   // Initial call of this OB
      Remanence : Bool;   // =True, if remanent data are available
   END_VAR
BEGIN

REGION Network 1
   // Read sensors
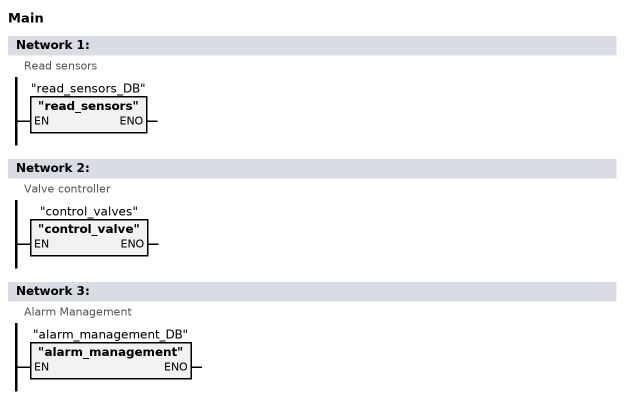
   RUNG wire#powerrail
      "read_sensors_DB"()
   END_RUNG
   // the same network as SCL:
   "read_sensors_DB"();   // "read_sensors"
END_REGION

REGION Network 2
   // Valve controller
   RUNG wire#powerrail
      "control_valves"()
   END_RUNG
   // the same network as SCL:
   "control_valves"();   // "control_valve"
END_REGION

REGION Network 3
   // Alarm Management
   RUNG wire#powerrail
      "alarm_management_DB"()
   END_RUNG
   // the same network as SCL:
   "alarm_management_DB"();   // "alarm_management"
END_REGION
END_ORGANIZATION_BLOCK

ORGANIZATION_BLOCK "temperature_controller"   // OB30, LAD, CyclicInterrupt
{ S7_Optimized_Access := 'TRUE' }
VERSION : 0.1
   VAR_INPUT
      Initial_Call : Bool;   // Initial call of this OB
      Event_Count : Int;   // Events discarded
   END_VAR
BEGIN

REGION Network 1: Temperature PID controller
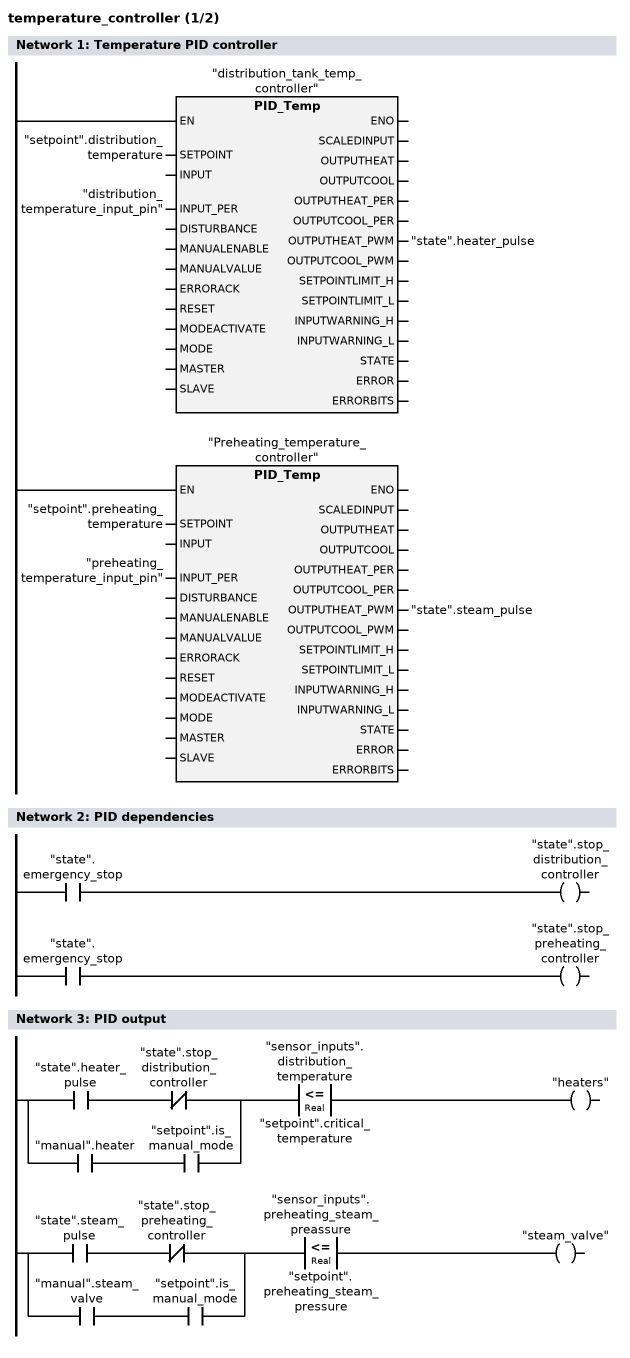
   "distribution_tank_temp_controller"(Setpoint := "setpoint".distribution_temperature,   // PID_Temp
                           Input_PER := "distribution_temperature_input_pin",
                           OutputHeat_PWM => "state".heater_pulse);
   "Preheating_temperature_controller"(Setpoint := "setpoint".preheating_temperature,   // PID_Temp
                           Input_PER := "preheating_temperature_input_pin",
                           OutputHeat_PWM => "state".steam_pulse);
END_REGION

REGION Network 2: PID dependencies
   RUNG wire#powerrail
      Contact( "state".emergency_stop )
      Coil( "state".stop_distribution_controller )
   END_RUNG
   RUNG wire#powerrail
      Contact( "state".emergency_stop )
      Coil( "state".stop_preheating_controller )
   END_RUNG
   // the same network as SCL:
   "state".stop_distribution_controller := "state".emergency_stop;
   "state".stop_preheating_controller := "state".emergency_stop;
END_REGION

REGION Network 3: PID output
   RUNG wire#powerrail
      Contact( "state".heater_pulse )
      I_Contact( "state".stop_distribution_controller )
      wire#w1
      { S7_Templates := "SrcType := Real" } LE_Contact(in1 := "sensor_inputs".distribution_temperature, in2 := "setpoint".critical_temperature)
      Coil( "heaters" )
   END_RUNG
   RUNG wire#powerrail
      Contact( "manual".heater )
      Contact( "setpoint".is_manual_mode )
   END_RUNG wire#w1
   RUNG wire#powerrail
      Contact( "state".steam_pulse )
      I_Contact( "state".stop_preheating_controller )
      wire#w2
      { S7_Templates := "SrcType := Real" } LE_Contact(in1 := "sensor_inputs".preheating_steam_preassure, in2 := "setpoint".preheating_steam_pressure)
      Coil( "steam_valve" )
   END_RUNG
   RUNG wire#powerrail
      Contact( "manual".steam_valve )
      Contact( "setpoint".is_manual_mode )
   END_RUNG wire#w2
   // the same network as SCL:
   "heaters" := (("state".heater_pulse AND NOT "state".stop_distribution_controller) OR ("manual".heater AND "setpoint".is_manual_mode)) AND ("sensor_inputs".distribution_temperature <= "setpoint".critical_temperature);
   "steam_valve" := (("state".steam_pulse AND NOT "state".stop_preheating_controller) OR ("manual".steam_valve AND "setpoint".is_manual_mode)) AND ("sensor_inputs".preheating_steam_preassure <= "setpoint".preheating_steam_pressure);
END_REGION

REGION Network 4: Trend Limit
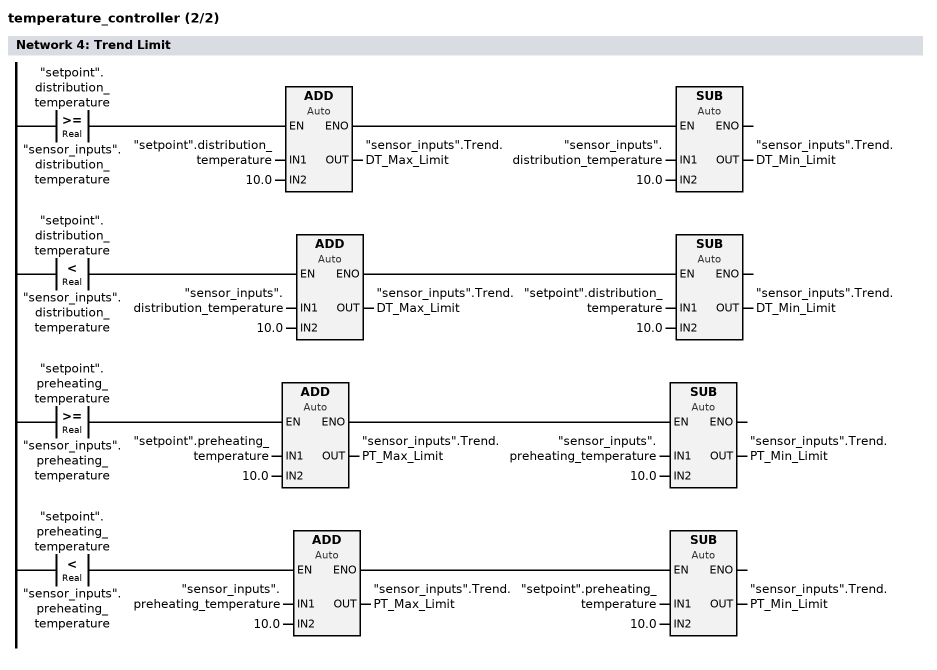
   RUNG wire#powerrail
      { S7_Templates := "SrcType := Real" } GE_Contact(in1 := "setpoint".distribution_temperature, in2 := "sensor_inputs".distribution_temperature)
      Add(in1 := "setpoint".distribution_temperature, in2 := 10.0, out => "sensor_inputs".Trend.DT_Max_Limit)
      Sub(in1 := "sensor_inputs".distribution_temperature, in2 := 10.0, out => "sensor_inputs".Trend.DT_Min_Limit)
   END_RUNG
   RUNG wire#powerrail
      { S7_Templates := "SrcType := Real" } LT_Contact(in1 := "setpoint".distribution_temperature, in2 := "sensor_inputs".distribution_temperature)
      Add(in1 := "sensor_inputs".distribution_temperature, in2 := 10.0, out => "sensor_inputs".Trend.DT_Max_Limit)
      Sub(in1 := "setpoint".distribution_temperature, in2 := 10.0, out => "sensor_inputs".Trend.DT_Min_Limit)
   END_RUNG
   RUNG wire#powerrail
      { S7_Templates := "SrcType := Real" } GE_Contact(in1 := "setpoint".preheating_temperature, in2 := "sensor_inputs".preheating_temperature)
      Add(in1 := "setpoint".preheating_temperature, in2 := 10.0, out => "sensor_inputs".Trend.PT_Max_Limit)
      Sub(in1 := "sensor_inputs".preheating_temperature, in2 := 10.0, out => "sensor_inputs".Trend.PT_Min_Limit)
   END_RUNG
   RUNG wire#powerrail
      { S7_Templates := "SrcType := Real" } LT_Contact(in1 := "setpoint".preheating_temperature, in2 := "sensor_inputs".preheating_temperature)
      Add(in1 := "sensor_inputs".preheating_temperature, in2 := 10.0, out => "sensor_inputs".Trend.PT_Max_Limit)
      Sub(in1 := "setpoint".preheating_temperature, in2 := 10.0, out => "sensor_inputs".Trend.PT_Min_Limit)
   END_RUNG
   // the same network as SCL:
   IF "setpoint".distribution_temperature >= "sensor_inputs".distribution_temperature THEN
       "sensor_inputs".Trend.DT_Max_Limit := "setpoint".distribution_temperature + 10.0;
       "sensor_inputs".Trend.DT_Min_Limit := "sensor_inputs".distribution_temperature - 10.0;
   END_IF;
   IF "setpoint".distribution_temperature < "sensor_inputs".distribution_temperature THEN
       "sensor_inputs".Trend.DT_Max_Limit := "sensor_inputs".distribution_temperature + 10.0;
       "sensor_inputs".Trend.DT_Min_Limit := "setpoint".distribution_temperature - 10.0;
   END_IF;
   IF "setpoint".preheating_temperature >= "sensor_inputs".preheating_temperature THEN
       "sensor_inputs".Trend.PT_Max_Limit := "setpoint".preheating_temperature + 10.0;
       "sensor_inputs".Trend.PT_Min_Limit := "sensor_inputs".preheating_temperature - 10.0;
   END_IF;
   IF "setpoint".preheating_temperature < "sensor_inputs".preheating_temperature THEN
       "sensor_inputs".Trend.PT_Max_Limit := "sensor_inputs".preheating_temperature + 10.0;
       "sensor_inputs".Trend.PT_Min_Limit := "setpoint".preheating_temperature - 10.0;
   END_IF;
END_REGION
END_ORGANIZATION_BLOCK

(* ===== HMI "HMI_RT_1" =====
system functions are stored by id; their names below are inferred from use
connection "HMI_Connection_1": ETHERNET, S7_1200_OMS

HMI tags "Default tag table"
   "Tag_ScreenNumber" : UInt, internal
   "ScreenNumber" : UInt, internal

HMI tags "I/O"
   "steam_preassure_sensor_pin" : Int = PLC steam_preassure_sensor_pin AT %IW96, 100 ms
   "preheating_pressure_sensor_pin" : Int = PLC preheating_pressure_sensor_pin AT %IW98, 100 ms
   "distribution_pressure_pin" : Int = PLC distribution_pressure_pin AT %IW100, 100 ms
   "preheating_temperature_input_pin" : Int = PLC preheating_temperature_input_pin AT %IW102, 100 ms
   "distribution_temperature_input_pin" : Int = PLC distribution_temperature_input_pin AT %IW112, 100 ms
   "heaters" : Bool = PLC heaters AT %Q0.0, 100 ms
   "washing_out" : Bool = PLC washing_out AT %Q0.1, 100 ms
   "washing_in" : Bool = PLC washing_in AT %Q0.2, 100 ms
   "washing_pump" : Bool = PLC washing_pump AT %Q0.3, 100 ms
   "preheating_upper_level_sensor" : Bool = PLC preheating_upper_level_sensor AT %I0.0, 100 ms
   "preheating_lower_level_sensor" : Bool = PLC preheating_lower_level_sensor AT %I0.1, 100 ms
   "distribution_upper_level_sensor" : Bool = PLC distribution_upper_level_sensor AT %I0.2, 100 ms
   "distribution_lower_level_sensor" : Bool = PLC distribution_lower_level_sensor AT %I0.3, 100 ms
   "steam_valve" : Bool = PLC steam_valve AT %Q0.4, 100 ms
   "preheating_tank_comp_air_valve" : Bool = PLC preheating_tank_comp_air_bubbling_valve AT %Q0.5, 100 ms
   "soft_water_inlet_valve" : Bool = PLC soft_water_inlet_valve AT %Q0.6, 100 ms
   "hot_water_transfer_valve" : Bool = PLC hot_water_transfer_valve AT %Q0.7, 100 ms
   "distribution_tank_comp_air_valve" : Bool = PLC distribution_tank_comp_air_bubbling_valve AT %Q1.0, 100 ms
   "distribution_valve" : Bool = PLC distribution_valve AT %Q1.1, 100 ms
   "preheating_vent" : Bool = PLC preheating_vent AT %Q8.0, 100 ms
   "distribution_vent" : Bool = PLC distribution_vent AT %Q8.1, 100 ms

HMI tags "Setpoint"
   "setpoint_distribution_temperature" : Real = PLC setpoint.distribution_temperature AT %DB3.DBD0, 100 ms
   "setpoint_distribution_temperature_tolerance" : Real = PLC setpoint.distribution_temperature_tolerance AT %DB3.DBD4, 100 ms
   "setpoint_preheating_temperature" : Real = PLC setpoint.preheating_temperature AT %DB3.DBD8, 100 ms
   "setpoint_preheating_temperature_tolerance" : Real = PLC setpoint.preheating_temperature_tolerance AT %DB3.DBD12, 100 ms
   "setpoint_distribution_tank_pressure" : Real = PLC setpoint.distribution_tank_pressure AT %DB3.DBD16, 100 ms
   "setpoint_preheating_tank_pressure" : Real = PLC setpoint.preheating_tank_pressure AT %DB3.DBD20, 100 ms
   "setpoint_preheating_steam_pressure" : Real = PLC setpoint.preheating_steam_pressure AT %DB3.DBD24, 100 ms
   "setpoint_preheating_steam_pressure_tolerance" : Real = PLC setpoint.preheating_steam_pressure_tolerance AT %DB3.DBD28, 100 ms
   "setpoint_preaheating_tank_pressure_tolerance" : Real = PLC setpoint.preaheating_tank_pressure_tolerance AT %DB3.DBD32, 100 ms
   "setpoint_distribution_tank_pressure_tolerance" : Real = PLC setpoint.distribution_tank_pressure_tolerance AT %DB3.DBD36, 100 ms
   "setpoint_is_manual_mode" : Bool = PLC setpoint.is_manual_mode AT %DB3.DBX40.0, 100 ms
   "read_sensors_DB_Steam_pressure_input_Calibration" : Real = PLC read_sensors_DB.Steam_pressure_input.Calibration, 1 s
   "read_sensors_DB_preheating_tank_pressure_input_Calibration" : Real = PLC read_sensors_DB.preheating_tank_pressure_input.Calibration, 1 s
   "read_sensors_DB_distribution_tank_pressure_input_Calibration" : Real = PLC read_sensors_DB.distribution_tank_pressure_input.Calibration, 1 s
   "read_sensors_DB_preheating_temperature_input_Calibration" : Real = PLC read_sensors_DB.preheating_temperature_input.Calibration, 1 s
   "read_sensors_DB_distribution_temperature_input_Calibration" : Real = PLC read_sensors_DB.distribution_temperature_input.Calibration, 1 s

HMI tags "State"
   "state_heater_pulse" : Bool = PLC state.heater_pulse AT %DB4.DBX0.0, 100 ms
   "state_distribution_tank_full" : Bool = PLC state.distribution_tank_full AT %DB4.DBX0.1, 100 ms
   "state_distribution_tank_empty" : Bool = PLC state.distribution_tank_empty AT %DB4.DBX0.2, 100 ms
   "state_preheating_tank_full" : Bool = PLC state.preheating_tank_full AT %DB4.DBX0.3, 100 ms
   "state_preheating_tank_empty" : Bool = PLC state.preheating_tank_empty AT %DB4.DBX0.4, 100 ms
   "state_stop_distribution_controller" : Bool = PLC state.stop_distribution_controller AT %DB4.DBX0.5, 100 ms
   "state_stop_preheating_controller" : Bool = PLC state.stop_preheating_controller AT %DB4.DBX0.6, 100 ms
   "state_steam_pulse" : Bool = PLC state.steam_pulse AT %DB4.DBX0.7, 100 ms
   "state_preheating_steam_pressure_high" : Bool = PLC state.preheating_steam_pressure_high AT %DB4.DBX1.0, 100 ms
   "state_preheating_tank_pressure_high" : Bool = PLC state.preheating_tank_pressure_high AT %DB4.DBX1.1, 100 ms
   "state_emergency_stop" : Bool = PLC state.emergency_stop AT %DB4.DBX1.2, 100 ms
   "state_preheating_temperature_in_range" : Bool = PLC state.preheating_temperature_in_range AT %DB4.DBX1.3, 100 ms
   "state_distribution_temperature_in_range" : Bool = PLC state.distribution_temperature_in_range AT %DB4.DBX1.4, 100 ms

HMI tags "Manual_Control"
   "manual_steam_valve" : Bool = PLC manual.steam_valve AT %DB7.DBX0.0, 100 ms
   "manual_preheating_tank_comp_air_valve" : Bool = PLC manual.preheating_tank_comp_air_valve AT %DB7.DBX0.1, 100 ms
   "manual_soft_water_inlet_valve" : Bool = PLC manual.soft_water_inlet_valve AT %DB7.DBX0.2, 100 ms
   "manual_hot_water_transfer_valve" : Bool = PLC manual.hot_water_transfer_valve AT %DB7.DBX0.3, 100 ms
   "manual_distribution_tank_comp_air_valve" : Bool = PLC manual.distribution_tank_comp_air_valve AT %DB7.DBX0.4, 100 ms
   "manual_distribution_valve" : Bool = PLC manual.distribution_valve AT %DB7.DBX0.5, 100 ms
   "manual_heater" : Bool = PLC manual.heater AT %DB7.DBX0.6, 100 ms
   "manual_preheating_vent" : Bool = PLC manual.preheating_vent AT %DB7.DBX0.7, 100 ms
   "manual_distribution_vent" : Bool = PLC manual.distribution_vent AT %DB7.DBX1.0, 100 ms

HMI tags "Alarm_limit"
   "alarm_limit_preheating_temperature_high_delay" : Time = PLC alarm_limit.preheating_temperature_high_delay AT %DB9.DBD44, 100 ms
   "alarm_limit_distribution_pressure_low" : Real = PLC alarm_limit.distribution_pressure_low AT %DB9.DBD48, 100 ms
   "alarm_limit_distribution_pressure_low_delay" : Time = PLC alarm_limit.distribution_pressure_low_delay AT %DB9.DBD52, 100 ms
   "alarm_limit_distribution_pressure_high" : Real = PLC alarm_limit.distribution_pressure_high AT %DB9.DBD56, 100 ms
   "alarm_limit_distribution_pressure_high_delay" : Time = PLC alarm_limit.distribution_pressure_high_delay AT %DB9.DBD60, 100 ms
   "alarm_limit_distribution_temperature_low" : Real = PLC alarm_limit.distribution_temperature_low AT %DB9.DBD64, 100 ms
   "alarm_limit_distribution_temperature_low_delay" : Time = PLC alarm_limit.distribution_temperature_low_delay AT %DB9.DBD68, 100 ms
   "alarm_limit_distribution_temperature_high" : Real = PLC alarm_limit.distribution_temperature_high AT %DB9.DBD72, 100 ms
   "alarm_limit_distribution_temperature_high_delay" : Time = PLC alarm_limit.distribution_temperature_high_delay AT %DB9.DBD76, 100 ms
   "alarm_limit_preheating_tank_empty" : Real = PLC alarm_limit.preheating_tank_empty AT %DB9.DBD80, 100 ms
   "alarm_limit_preheating_tank_empty_delay" : Time = PLC alarm_limit.preheating_tank_empty_delay AT %DB9.DBD84, 100 ms
   "alarm_limit_distribution_tank_empty" : Real = PLC alarm_limit.distribution_tank_empty AT %DB9.DBD88, 100 ms
   "alarm_limit_distribution_tank_empty_delay" : Time = PLC alarm_limit.distribution_tank_empty_delay AT %DB9.DBD92, 100 ms
   "alarm_limit_steam_pressure_low" : Real = PLC alarm_limit.steam_pressure_low AT %DB9.DBD0, 1 s
   "alarm_limit_steam_pressure_low_delay" : Time = PLC alarm_limit.steam_pressure_low_delay AT %DB9.DBD4, 1 s
   "alarm_limit_steam_pressure_high" : Real = PLC alarm_limit.steam_pressure_high AT %DB9.DBD8, 1 s
   "alarm_limit_steam_pressure_high_delay" : Time = PLC alarm_limit.steam_pressure_high_delay AT %DB9.DBD12, 1 s
   "alarm_limit_preaheating_tank_pressure_low" : Real = PLC alarm_limit.preaheating_tank_pressure_low AT %DB9.DBD16, 1 s
   "alarm_limit_preaheating_tank_pressure_low_delay" : Time = PLC alarm_limit.preaheating_tank_pressure_low_delay AT %DB9.DBD20, 1 s
   "alarm_limit_preaheating_tank_pressure_high" : Real = PLC alarm_limit.preaheating_tank_pressure_high AT %DB9.DBD24, 1 s
   "alarm_limit_preaheating_tank_pressure_high_delay" : Time = PLC alarm_limit.preaheating_tank_pressure_high_delay AT %DB9.DBD28, 1 s
   "alarm_limit_preheating_temperature_low" : Real = PLC alarm_limit.preheating_temperature_low AT %DB9.DBD32, 1 s
   "alarm_limit_preheating_temperature_low_delay" : Time = PLC alarm_limit.preheating_temperature_low_delay AT %DB9.DBD36, 1 s
   "alarm_limit_preheating_temperature_high" : Real = PLC alarm_limit.preheating_temperature_high AT %DB9.DBD40, 1 s

HMI tags "Alarm"
   "alarm" : Int = PLC alarm AT %MW2, 100 ms
   "steam_pressure_low" : Bool = PLC steam_pressure_low AT %M2.0, 100 ms
   "preaheating_tank_pressure_low" : Bool = PLC preaheating_tank_pressure_low AT %M2.2, 100 ms
   "preaheating_tank_pressure_high" : Bool = PLC preaheating_tank_pressure_high AT %M2.3, 100 ms
   "preheating_temperature_low" : Bool = PLC preheating_temperature_low AT %M2.4, 100 ms
   "preheating_temperature_high" : Bool = PLC preheating_temperature_high AT %M2.5, 100 ms
   "steam_pressure_high" : Bool = PLC steam_pressure_high AT %M2.1, 100 ms
   "distribution_pressure_low" : Bool = PLC distribution_pressure_low AT %M2.6, 100 ms
   "distribution_pressure_high" : Bool = PLC distribution_pressure_high AT %M2.7, 100 ms
   "distribution_temperature_low" : Bool = PLC distribution_temperature_low AT %M3.0, 100 ms
   "distribution_temperature_high" : Bool = PLC distribution_temperature_high AT %M3.1, 100 ms
   "preheating_tank_empty" : Bool = PLC preheating_tank_empty AT %M3.2, 100 ms
   "distribution_tank_empty" : Bool = PLC distribution_tank_empty AT %M3.3, 100 ms

HMI tags "Sensor_Inputs"
   "sensor_inputs_preheating_steam_preassure" : Real = PLC sensor_inputs.preheating_steam_preassure AT %DB1.DBD0, 100 ms
   "sensor_inputs_preheating_tank_pressure" : Real = PLC sensor_inputs.preheating_tank_pressure AT %DB1.DBD4, 100 ms
   "sensor_inputs_distribution_tank_pressure" : Real = PLC sensor_inputs.distribution_tank_pressure AT %DB1.DBD8, 100 ms
   "sensor_inputs_preheating_temperature" : Real = PLC sensor_inputs.preheating_temperature AT %DB1.DBD12, 100 ms
   "sensor_inputs_distribution_temperature" : Real = PLC sensor_inputs.distribution_temperature AT %DB1.DBD16, 100 ms
   "sensor_inputs_Trend_DT_Max_Limit" : Real = PLC sensor_inputs.Trend.DT_Max_Limit AT %DB1.DBD20, 1 s
   "sensor_inputs_Trend_DT_Min_Limit" : Real = PLC sensor_inputs.Trend.DT_Min_Limit AT %DB1.DBD24, 1 s
   "sensor_inputs_Trend_PT_Max_Limit" : Real = PLC sensor_inputs.Trend.PT_Max_Limit AT %DB1.DBD28, 1 s
   "sensor_inputs_Trend_PT_Min_Limit" : Real = PLC sensor_inputs.Trend.PT_Min_Limit AT %DB1.DBD32, 1 s

HMI tags "PID_tuning"
   "Preheating_temperature_controller_Retain_CtrlParams_Heat" : PID_TempControlParams = PLC Preheating_temperature_controller.Retain.CtrlParams.Heat, 1 s
   "Preheating_temperature_controller_Retain_CtrlParams_Cool" : PID_TempControlParams = PLC Preheating_temperature_controller.Retain.CtrlParams.Cool, 1 s
   "distribution_tank_temp_controller_Retain_CtrlParams_Heat" : PID_TempControlParams = PLC distribution_tank_temp_controller.Retain.CtrlParams.Heat, 1 s
   "distribution_tank_temp_controller_Retain_CtrlParams_Cool" : PID_TempControlParams = PLC distribution_tank_temp_controller.Retain.CtrlParams.Cool, 1 s

discrete alarms
   1: 'Steam pressure has reached low level', class Errors, trigger "alarm" bit 0
   2: 'Steam pressure has reached high level', class Errors, trigger "alarm" bit 1
   3: 'Heating tank pressure has reached low level', class Errors, trigger "alarm" bit 2
   4: 'Heating tank pressure has reached high level', class Errors, trigger "alarm" bit 3
   5: 'Heating tank temperature has reached low level', class Errors, trigger "alarm" bit 4
   6: 'Heating tank temperature has reached high level', class Errors, trigger "alarm" bit 5
   7: 'Distribution tank pressure has reached low level', class Errors, trigger "alarm" bit 6
   8: 'Distribution tank pressure has reached high level', class Errors, trigger "alarm" bit 7
   9: 'Distribution tank temperature has reached low level', class Errors, trigger "alarm" bit 8
   10: 'Distribution tank temperature has reached high level', class Errors, trigger "alarm" bit 9

text list "V_HCA": 0 'Auto'; 1 'Manual'

screen "Home" 800x480
   on GenerateScreen: SetTag("Tag_ScreenNumber", 1)
   TextField "Text field_1" at 45,210 size 511x112; Text 'HOT WATER GENERATION PLANT'
   GraphicView "Graphic view_2" at 510,134 size 254x279; Picture "Graphic_45"
   Button "Button_1" at 520,196 size 224x149; TextOff 'Text'
      on Click: ActivateScreen("Overview", 0); SetTag("ScreenNumber", 2)
   GraphicView "Graphic view_1" at 10,1 size 149x57; Picture "Renata-Blue"
   Button "Button_2" at 170,2 size 480x60; TextOff 'Renata Limited (Mirpur Site)'
   DateTimeField "HmiScreenItemData" at 670,30 size 119x24
   DateTimeField "HmiScreenItemData_1" at 676,6 size 113x24

screen "Overview" 800x480, template "Lower Button"
   GraphicView "Preheating tank outer hull" at 404,124 size 170x193; Picture "Graphic_4"
   GraphicView "Preheating tank inner hull" at 418,133 size 140x168; Picture "Graphic_4"
   GraphicView "Preheating tank outer hull_1" at 109,124 size 170x193; Picture "Graphic_4"
   GraphicView "Preheating tank inner hull_1" at 123,133 size 140x168; Picture "Graphic_4"
   GraphicView "V-HSW Off" at 261,79 size 45x35; Picture "Graphic_37"
      Visibility <- "soft_water_inlet_valve"
   GraphicView "V-HSW On" at 261,79 size 45x35; Picture "Graphic_38"
      Visibility <- "soft_water_inlet_valve"
   GraphicView "Off" at 141,75 size 35x45; Picture "Graphic_41"
      Visibility <- "preheating_tank_comp_air_valve"
   GraphicView "On" at 141,75 size 35x45; Picture "Graphic_40"
      Visibility <- "preheating_tank_comp_air_valve"
   Button "Button_4" at 255,323 size 85x40; TextOff 'Text'
   IOField "I/O field_2" at 260,339 size 55x23; FormatPattern 999.9
      ProcessValue <- "sensor_inputs_preheating_temperature"
   TextField "Text field_8" at 273,320 size 51x21; Text 'TS-H01'
   TextField "Text field_9" at 314,338 size 20x21; Text '◦c'
   Button "Button_7" at 186,139 size 85x40; TextOff 'Text'
   IOField "I/O field_4" at 187,155 size 55x23; FormatPattern 999.9
      ProcessValue <- "sensor_inputs_preheating_tank_pressure"
   TextField "Text field_14" at 206,136 size 51x21; Text 'PS-H01'
   TextField "Text field_15" at 242,154 size 35x21; Text 'bar'
   Button "Button_5" at 23,110 size 85x40; TextOff 'Text'
   IOField "I/O field_1" at 24,126 size 55x23; FormatPattern 999.9
      ProcessValue <- "sensor_inputs_preheating_steam_preassure"
   TextField "Text field_10" at 43,107 size 51x21; Text 'PS-H02'
   TextField "Text field_11" at 79,125 size 35x21; Text 'bar'
   Button "Button_6" at 551,323 size 85x40; TextOff 'Text'
   IOField "I/O field_3" at 556,339 size 55x23; FormatPattern 999.9
      ProcessValue <- "sensor_inputs_distribution_temperature"
   TextField "Text field_12" at 569,320 size 52x21; Text 'TS-D01'
   TextField "Text field_13" at 610,338 size 20x21; Text '◦c'
   Button "Button_8" at 400,171 size 85x40; TextOff 'Text'
   IOField "I/O field_5" at 401,187 size 55x23; FormatPattern 999.9
      ProcessValue <- "sensor_inputs_distribution_tank_pressure"
   TextField "Text field_16" at 420,168 size 52x21; Text 'PS-D01'
   TextField "Text field_17" at 456,186 size 35x21; Text 'bar'
   GraphicView "Off_1" at 515,70 size 35x45; Picture "Graphic_41"
      Visibility <- "distribution_tank_comp_air_valve"
   GraphicView "On_1" at 515,70 size 35x45; Picture "Graphic_40"
      Visibility <- "distribution_tank_comp_air_valve"
   GraphicView "V-HWT Off" at 256,375 size 45x35; Picture "Graphic_37"
      Visibility <- "hot_water_transfer_valve"
   GraphicView "V-HWT On" at 256,375 size 45x35; Picture "Graphic_38"
      Visibility <- "hot_water_transfer_valve"
   GraphicView "V-D Off" at 552,375 size 45x35; Picture "Graphic_37"
      Visibility <- "distribution_valve"
   GraphicView "V-D On" at 552,375 size 45x35; Picture "Graphic_38"
      Visibility <- "distribution_valve"
   GraphicView "V-SM Off" at 56,213 size 45x35; Picture "Graphic_37"
      Visibility <- "steam_valve"
   GraphicView "V-SM On" at 56,213 size 45x35; Picture "Graphic_38"
      Visibility <- "steam_valve"
   GraphicView "Off_2" at 187,95 size 25x30; Picture "Graphic_41"
      Visibility <- "preheating_vent"
   GraphicView "On_2" at 187,95 size 25x30; Picture "Graphic_40"
      Visibility <- "preheating_vent"
   GraphicView "Off_3" at 477,95 size 25x30; Picture "Graphic_41"
      Visibility <- "distribution_vent"
   GraphicView "On_3" at 477,95 size 25x30; Picture "Graphic_40"
      Visibility <- "distribution_vent"
   Button "Button_17" at 694,6 size 100x67; TextOff 'Operating Mode'
      on Click: SetTag("ScreenNumber", 1)
      on Release: ActivateScreen("Home", 0)
      Appearance <- "ScreenNumber"
   GraphicView "Graphic view_9" at 427,50 size 32x32; Picture "Graphic_19"
   GraphicView "Graphic view_14" at 40,218 size 80x30; Picture "Graphic_22"
   Line "Line_61" at 44,232 size 72x0
      Visibility <- "steam_valve"
   Group "Group" at 109,124 size 170x193; Picture "Graphic_4"
   GraphicView "Graphic view_13" at 140,63 size 30x80; Picture "Graphic_16"
      Appearance <- "preheating_upper_level_sensor"
   Line "Line_60" at 154,66 size 0x72
      Visibility <- "preheating_tank_comp_air_valve"
   GraphicView "Graphic view_16" at 187,333 size 65x34; Picture "Graphic_9"
   Group "Preheating tank" at 404,124 size 170x193; Picture "Graphic_4"
   GraphicView "Graphic view_6" at 176,312 size 30x70; Picture "Graphic_16"
   GraphicView "Graphic view_11" at 175,380 size 32x32; Picture "Graphic_21"
   GraphicView "Graphic view_12" at 203,381 size 160x30; Picture "Graphic_22"
   GraphicView "Graphic view_10" at 361,380 size 32x32; Picture "Graphic_20"
   GraphicView "Graphic view_1" at 362,78 size 30x305; Picture "Graphic_16"
   GraphicView "Graphic view_7" at 362,50 size 32x32; Picture "Graphic_17"
   GraphicView "Graphic view_2" at 390,51 size 45x30; Picture "Graphic_22"
   GraphicView "Graphic view_3" at 428,78 size 30x68; Picture "Graphic_16"
   GraphicView "Graphic view_4" at 218,112 size 30x30; Picture "Graphic_16"
   GraphicView "Graphic view_5" at 217,84 size 32x32; Picture "Graphic_17"
   GraphicView "Graphic view_8" at 245,85 size 80x30; Picture "Graphic_22"
   GraphicView "Graphic view_17" at 477,333 size 65x34; Picture "Graphic_9"
   GraphicView "Graphic view_19" at 466,312 size 30x70; Picture "Graphic_16"
   GraphicView "Graphic view_20" at 465,380 size 32x32; Picture "Graphic_21"
   GraphicView "Graphic view_21" at 493,381 size 160x30; Picture "Graphic_22"
   GraphicView "Graphic view_18" at 513,58 size 30x86; Picture "Graphic_16"
   Button "Button_1" at 28,17 size 150x25; TextOff 'Compressed Air'
   Group "Group_5" at 147,54 size 12x6
   Button "Button_2" at 260,38 size 110x25; TextOff 'Soft Water'
   Group "Group_6" at 315,84 size 12x6
   TextField "Text field_5" at 152,215 size 71x40; Text 'Heating Tank'
   TextField "Text field_6" at 437,215 size 107x40; Text 'Distribution Tank'
   Button "Button_3" at 675,383 size 110x25; TextOff 'Hot Water'
   Group "Group_7" at 668,389 size 6x12
   GraphicView "Graphic view_23" at 113,115 size 25x32; Picture "Graphic_14"
   GraphicView "Graphic view_25" at 160,147 size 25x32; Picture "Graphic_14"
   GraphicView "Graphic view_27" at 488,147 size 25x32; Picture "Graphic_14"
   Group "Group_9" at 23,107 size 91x43
   Group "Group_10" at 255,320 size 85x43
   Group "Group_11" at 551,320 size 85x43
   Group "Group_12" at 400,168 size 91x43
   Button "Button_9" at 496,12 size 150x25; TextOff 'Compressed Air'
   Group "Group_13" at 521,49 size 12x6
   TextField "Text field_2" at 271,203 size 50x21; Text 'LS-H02'
   Circle "Circle_1" at 273,223 size 24x24
      Appearance <- "preheating_lower_level_sensor"
   TextField "Text field_1" at 271,152 size 50x21; Text 'LS-H01'
   Circle "Circle_2" at 273,172 size 24x24
      Appearance <- "preheating_upper_level_sensor"
   TextField "Text field_3" at 567,235 size 51x21; Text 'LS-D02'
   Circle "Circle_3" at 569,255 size 24x24
      Appearance <- "distribution_lower_level_sensor"
   TextField "Text field_4" at 567,147 size 51x21; Text 'LS-D01'
   Circle "Circle_4" at 569,167 size 24x24
      Appearance <- "distribution_upper_level_sensor"
   Group "V-HCA" at 141,75 size 35x45; Picture "Graphic_41"
   Group "Group_1" at 34,242 size 12x6
   Group "V-SM" at 56,213 size 45x35; Picture "Graphic_37"
   Button "Button_11" at 16,268 size 80x25; TextOff 'Steam'
   Button "Button_10" at 133,67 size 50x60; TextOff 'Text'
      on Release: function_efd93a16("V-HCA", 200, 100, -1, 0, 1)
   Button "Button_14" at 49,206 size 60x50; TextOff 'Text'
      on Release: function_efd93a16("V-SM", 80, 250, -1, 0, 1)
   Line "Line_65" at 301,395 size 62x0
      Visibility <- "hot_water_transfer_valve"
   Line "Line_66" at 367,389 size 6x5
      Visibility <- "hot_water_transfer_valve"
   Line "Line_67" at 376,78 size 0x308
      Visibility <- "hot_water_transfer_valve"
   Line "Line_68" at 377,67 size 6x8
      Visibility <- "hot_water_transfer_valve"
   Line "Line_69" at 387,65 size 45x0
      Visibility <- "hot_water_transfer_valve"
   Line "Line_70" at 435,67 size 5x5
      Visibility <- "hot_water_transfer_valve"
   Line "Line_71" at 442,76 size 0x66
      Visibility <- "hot_water_transfer_valve"
   Line "Line_75" at 597,395 size 50x0
      Visibility <- "distribution_valve"
   Group "V-HWT" at 256,375 size 45x35; Picture "Graphic_37"
   Button "Button_15" at 249,367 size 60x50; TextOff 'Text'
      on Release: function_efd93a16("V-HWT", 320, 250, -1, 3, 1)
   Group "V-D" at 552,375 size 45x35; Picture "Graphic_37"
   Button "Button_16" at 544,366 size 60x50; TextOff 'Text'
      on Release: function_efd93a16("V-D", 600, 250, -1, 2, 1)
   Line "Line_76" at 232,112 size 0x30
      Visibility <- "soft_water_inlet_valve"
   Line "Line_77" at 233,100 size 7x8
      Visibility <- "soft_water_inlet_valve"
   Line "Line_78" at 243,99 size 75x0
      Visibility <- "soft_water_inlet_valve"
   Group "Group_8" at 186,136 size 91x43
   Group "Group_2" at 261,79 size 45x35; Picture "Graphic_37"
   Button "Button_13" at 254,69 size 60x50; TextOff 'Text'
      on Release: function_efd93a16("V-HSW", 300, 100, -1, 1, 1)
   Line "Line_79" at 527,61 size 0x78
      Visibility <- "distribution_tank_comp_air_valve"
   Group "V-DCA" at 515,70 size 35x45; Picture "Graphic_41"
   Button "Button_12" at 513,62 size 50x60; TextOff 'Text'
      on Release: function_efd93a16("V-DCA", 550, 100, -1, 2, 1)
   SymbolicIOField "Symbolic I/O field_1" at 701,42 size 90x25; TextOn '1'; TextOff '0'; TextList "V_HCA"; Authorization "User administration"
      ProcessValue <- "setpoint_is_manual_mode"
   GraphicView "Graphic view_15" at 186,84 size 25x55; Picture "Graphic_16"
      Appearance <- "preheating_upper_level_sensor"
   Line "Line_80" at 198,87 size 0x48
      Visibility <- "preheating_vent"
   Group "V-HCA_1" at 187,95 size 25x30; Picture "Graphic_41"
   GraphicView "Graphic view_22" at 474,84 size 25x55; Picture "Graphic_16"
      Appearance <- "preheating_upper_level_sensor"
   Line "Line_81" at 485,87 size 0x48
      Visibility <- "distribution_vent"
   Group "V-HCA_2" at 477,95 size 25x30; Picture "Graphic_41"
   Button "Button_18" at 181,85 size 40x52; TextOff 'Text'
      on Release: function_efd93a16("V-PV", 250, 100, -1, 0, 1)
   Button "Button_19" at 180,39 size 70x25; TextOff 'Vent'
   Group "Group_3" at 191,66 size 12x6
   Button "Button_20" at 444,39 size 70x25; TextOff 'Vent'
   Group "Group_4" at 480,66 size 12x6
   Button "Button_21" at 468,84 size 40x52; TextOff 'Text'
      on Release: function_efd93a16("V-DV", 500, 100, -1, 0, 1)

screen "Rough" 800x480
   GraphicView "Preheating tank outer hull" at 181,19 size 170x193; Picture "Graphic_4"
   GraphicView "Preheating tank inner hull" at 195,28 size 140x168; Picture "Graphic_4"
   Group "Preheating tank" at 181,19 size 170x193; Picture "Graphic_4"
   GraphicView "Graphic view_2" at 320,343 size 60x38; Picture "Graphic_11"
   GraphicView "Graphic view_3" at 321,299 size 53x42; Picture "Graphic_12"
   GraphicView "Graphic view_4" at 384,313 size 33x60; Picture "Graphic_14"
   GraphicView "Graphic view_5" at 263,341 size 30x38; Picture "Graphic_15"
   GraphicView "Graphic view_7" at 541,194 size 75x75; Picture "Graphic_17"
   GraphicView "Graphic view_9" at 557,146 size 75x75; Picture "Graphic_19"
   GraphicView "Graphic view_10" at 517,247 size 75x75; Picture "Graphic_20"
   GraphicView "Graphic view_11" at 496,196 size 75x75; Picture "Graphic_21"
   GraphicView "Graphic view_12" at 550,106 size 75x75; Picture "Graphic_22"
   GraphicView "Graphic view_13" at 550,351 size 75x75; Picture "Graphic_24"
   GraphicView "Graphic view_14" at 529,373 size 75x75; Picture "Graphic_25"
   GraphicView "Graphic view_15" at 536,291 size 75x75; Picture "Graphic_26"
   GraphicView "Graphic view_16" at 554,273 size 75x75; Picture "Graphic_27"
   GraphicView "Graphic view_8" at 479,348 size 75x75; Picture "Graphic_18"
   GraphicView "Graphic view_17" at 648,65 size 121x120; Picture "Graphic_32"
   GraphicView "Graphic view_20" at 658,148 size 121x120; Picture "Graphic_34"
   GraphicView "Graphic view_21" at 635,118 size 121x120; Picture "Graphic_31"
   GraphicView "Graphic view_6" at 318,390 size 60x38; Picture "Graphic_11"
   GraphicView "Graphic view_18" at 263,408 size 47x43; Picture "Graphic_36"
   GraphicView "Graphic view_19" at 204,375 size 59x51; Picture "Graphic_35"
   GraphicView "Graphic view_22" at 121,311 size 83x69; Picture "Graphic_37"
   GraphicView "Graphic view_23" at 121,375 size 45x35; Picture "Graphic_38"
   GraphicView "Preheating tank outer hull_1" at 4,18 size 170x193; Picture "Graphic_4"
   GraphicView "Preheating tank inner hull_1" at 18,27 size 140x168; Picture "Graphic_4"
   GraphicView "Graphic view_28" at 228,321 size 35x45; Picture "Graphic_40"
   Button "Button_18" at 675,9 size 120x55; TextOff 'Operating Mode'
   SymbolicIOField "Symbolic I/O field_1" at 554,28 size 110x25; TextOn '1'; TextOff '0'; TextList "V_HCA"; Authorization "User administration"
      ProcessValue <- "setpoint_is_manual_mode"

Template "Lower Button" 800x480
   Button "Button_4" at 2,440 size 132x40; TextOff 'Home'
      on Release: ActivateScreen("Home", 0)
      on Click: SetTag("ScreenNumber", 1)
      Appearance <- "ScreenNumber"
   Button "Button_5" at 135,440 size 132x40; TextOff 'Overview'
      on Release: ActivateScreen("Overview", 0)
      Appearance <- "ScreenNumber"
      on Click: SetTag("ScreenNumber", 2)
   Button "Button_6" at 268,440 size 132x40; TextOff 'System Setpoints'; Authorization "User administration"
      on Release: ActivateScreen("System_Setpoints", 0)
      on Click: SetTag("ScreenNumber", 3)
      Appearance <- "ScreenNumber"
   Button "Button_7" at 401,440 size 132x40; TextOff 'Analog Control'
      on Release: ActivateScreen("Analog_Control", 0)
      on Click: SetTag("ScreenNumber", 4)
      Appearance <- "ScreenNumber"
   Button "Button_8" at 667,440 size 132x40; TextOff 'Alarm'
      on Release: ActivateScreen("Alarm", 0)
      on Click: SetTag("ScreenNumber", 6)
      Appearance <- "ScreenNumber"
   Button "Button_1" at 534,440 size 132x40; TextOff 'Trend'
      on Click: SetTag("ScreenNumber", 5)
      on Release: ActivateScreen("Trend", 0)
      Appearance <- "ScreenNumber"

PopupScreen "V-HCA" 185x95
   GraphicView "V-HCA Off" at 126,6 size 45x35; Picture "Graphic_37"
      Visibility <- "preheating_tank_comp_air_valve"
   GraphicView "V-HCA On" at 126,6 size 45x35; Picture "Graphic_38"
      Visibility <- "preheating_tank_comp_air_valve"
   Button "Button_1" at 2,3 size 180x40; TextOff 'Heating Tank Cmp Air Valve'
   Button "Button_5" at 2,42 size 180x50; TextOff 'Manual Operation'
   Button "Button_6" at 5,57 size 85x32; TextOff 'Start'
      on Press: SetBit("manual_preheating_tank_comp_air_valve")
   Button "Button_7" at 94,57 size 85x32; TextOff 'Stop'
      on Press: ResetBit("manual_preheating_tank_comp_air_valve")
   Group "V-HCA" at 126,6 size 45x35; Picture "Graphic_37"

PopupScreen "V-HSW" 185x95
   GraphicView "V-HSW Off" at 124,6 size 45x35; Picture "Graphic_37"
      Visibility <- "soft_water_inlet_valve"
   GraphicView "V-HSW On" at 124,6 size 45x35; Picture "Graphic_38"
      Visibility <- "soft_water_inlet_valve"
   Button "Button_1" at 2,3 size 180x40; TextOff 'Soft Water Valve'
   Button "Button_5" at 2,42 size 180x50; TextOff 'Manual Operation'
   Button "Button_6" at 5,57 size 85x32; TextOff 'Start'
      on Press: SetBit("manual_soft_water_inlet_valve")
   Button "Button_7" at 94,57 size 85x32; TextOff 'Stop'
      on Press: ResetBit("manual_soft_water_inlet_valve")
   Group "V-HWT_1" at 124,6 size 45x35; Picture "Graphic_37"

PopupScreen "V-DCA" 185x95
   GraphicView "V-DCA Off" at 126,6 size 45x35; Picture "Graphic_37"
      Visibility <- "distribution_tank_comp_air_valve"
   GraphicView "V-DCA On" at 126,6 size 45x35; Picture "Graphic_38"
      Visibility <- "distribution_tank_comp_air_valve"
   Button "Button_1" at 2,3 size 180x40; TextOff 'Distribution Tank Cmp Air Valve'
   Button "Button_5" at 2,42 size 180x50; TextOff 'Manual Operation'
   Button "Button_6" at 5,57 size 85x32; TextOff 'Start'
      on Press: SetBit("manual_distribution_tank_comp_air_valve")
   Button "Button_7" at 94,57 size 85x32; TextOff 'Stop'
      on Press: ResetBit("manual_distribution_tank_comp_air_valve")
   Group "V-DCA" at 126,6 size 45x35; Picture "Graphic_37"

PopupScreen "V-SM" 185x95
   GraphicView "V-SM Off" at 126,6 size 45x35; Picture "Graphic_37"
      Visibility <- "steam_valve"
   GraphicView "V-SM On" at 126,6 size 45x35; Picture "Graphic_38"
      Visibility <- "steam_valve"
   Button "Button_1" at 2,3 size 180x40; TextOff 'Steam Main Valve'
   Button "Button_5" at 2,42 size 180x50; TextOff 'Manual Operation'
   Button "Button_6" at 5,57 size 85x32; TextOff 'Start'
      on Press: SetBit("manual_steam_valve")
   Button "Button_7" at 94,57 size 85x32; TextOff 'Stop'
      on Press: ResetBit("manual_steam_valve")
   Group "V-SM" at 126,6 size 45x35; Picture "Graphic_37"

PopupScreen "V-D" 185x95
   GraphicView "V-D Off" at 126,6 size 45x35; Picture "Graphic_37"
      Visibility <- "distribution_valve"
   GraphicView "V-D On" at 126,6 size 45x35; Picture "Graphic_38"
      Visibility <- "distribution_valve"
   Button "Button_1" at 2,3 size 180x40; TextOff 'Distribution Valve'
   Button "Button_5" at 2,42 size 180x50; TextOff 'Manual Operation'
   Button "Button_6" at 5,57 size 85x32; TextOff 'Start'
      on Press: SetBit("manual_distribution_valve")
   Button "Button_7" at 94,57 size 85x32; TextOff 'Stop'
      on Press: ResetBit("manual_distribution_valve")
   Group "V-D" at 126,6 size 45x35; Picture "Graphic_37"

PopupScreen "V-HWT" 185x95
   GraphicView "V-HWT Off" at 126,6 size 45x35; Picture "Graphic_37"
      Visibility <- "hot_water_transfer_valve"
   GraphicView "V-HWT On" at 126,6 size 45x35; Picture "Graphic_38"
      Visibility <- "hot_water_transfer_valve"
   Button "Button_1" at 2,3 size 180x40; TextOff 'Hot Water Transfer'
   Button "Button_5" at 2,42 size 180x50; TextOff 'Manual Operation'
   Button "Button_6" at 5,57 size 85x32; TextOff 'Start'
      on Press: SetBit("manual_hot_water_transfer_valve")
   Button "Button_7" at 94,57 size 85x32; TextOff 'Stop'
      on Press: ResetBit("manual_hot_water_transfer_valve")
   Group "V-HWT" at 126,6 size 45x35; Picture "Graphic_37"

screen "Analog_Control" 800x480, template "Lower Button"
   Button "Button_15" at 2,243 size 216x36; TextOff 'Text'
   Button "Button_14" at 2,202 size 216x36; TextOff 'Text'
   Button "Button_13" at 2,161 size 216x36; TextOff 'Text'
   Button "Button_12" at 2,120 size 216x36; TextOff 'Text'
   Button "Button_11" at 2,79 size 216x36; TextOff 'Text'
   Button "Button_1" at 222,25 size 245x50; TextOff 'High Alarm'
   Button "Button_2" at 222,49 size 90x25; TextOff 'Setpoint'
   Button "Button_4" at 312,49 size 100x25; TextOff 'Delay time (s)'
   Button "Button_7" at 411,49 size 55x25; TextOff 'Status'
   Button "Button_3" at 468,25 size 245x50; TextOff 'Low Alarm'
   Button "Button_5" at 468,49 size 90x25; TextOff 'Setpoint'
   Button "Button_6" at 558,49 size 100x25; TextOff 'Delay time (s)'
   Button "Button_10" at 657,49 size 55x25; TextOff 'Status'
   Button "Button_9" at 714,25 size 80x50; TextOff 'Process Value'
   Button "Button_8" at 221,78 size 574x203; TextOff 'Text'
   IOField "I/O field_5" at 225,80 size 85x35; FormatPattern 999.9
      ProcessValue <- "alarm_limit_steam_pressure_high"
   TextField "Text field_16" at 4,84 size 127x21; Text 'Steam Pressure'
   IOField "I/O field_1" at 315,80 size 95x35; FormatPattern 9999
      ProcessValue <- "alarm_limit_steam_pressure_high_delay"
   Circle "Circle_1" at 423,80 size 30x30
      Appearance <- "steam_pressure_high"
   IOField "I/O field_2" at 225,120 size 85x35; FormatPattern 999.9
      ProcessValue <- "alarm_limit_preaheating_tank_pressure_high"
   IOField "I/O field_3" at 225,160 size 85x35; FormatPattern 999.9
      ProcessValue <- "alarm_limit_distribution_pressure_high"
   IOField "I/O field_4" at 225,200 size 85x35; FormatPattern 999.9
      ProcessValue <- "alarm_limit_preheating_temperature_high"
   IOField "I/O field_6" at 225,240 size 85x35; FormatPattern 999.9
      ProcessValue <- "alarm_limit_distribution_temperature_high"
   IOField "I/O field_7" at 315,120 size 95x35; FormatPattern 9999
      ProcessValue <- "alarm_limit_preaheating_tank_pressure_high_delay"
   IOField "I/O field_8" at 315,160 size 95x35; FormatPattern 9999
      ProcessValue <- "alarm_limit_distribution_pressure_high_delay"
   IOField "I/O field_9" at 315,200 size 95x35; FormatPattern 9999
      ProcessValue <- "alarm_limit_preheating_temperature_high_delay"
   IOField "I/O field_10" at 315,240 size 95x35; FormatPattern 9999
      ProcessValue <- "alarm_limit_distribution_temperature_high_delay"
   Circle "Circle_2" at 423,120 size 30x30
      Appearance <- "preaheating_tank_pressure_high"
   IOField "I/O field_11" at 473,80 size 85x35; FormatPattern 999.9
      ProcessValue <- "alarm_limit_steam_pressure_low"
   IOField "I/O field_12" at 563,80 size 95x35; FormatPattern 9999
      ProcessValue <- "alarm_limit_steam_pressure_low_delay"
   Circle "Circle_6" at 671,80 size 30x30
      Appearance <- "steam_pressure_low"
   IOField "I/O field_13" at 473,120 size 85x35; FormatPattern 999.9
      ProcessValue <- "alarm_limit_preaheating_tank_pressure_low"
   IOField "I/O field_14" at 473,160 size 85x35; FormatPattern 999.9
      ProcessValue <- "alarm_limit_distribution_pressure_low"
   IOField "I/O field_15" at 473,200 size 85x35; FormatPattern 999.9
      ProcessValue <- "alarm_limit_preheating_temperature_low"
   IOField "I/O field_16" at 473,240 size 85x35; FormatPattern 999.9
      ProcessValue <- "alarm_limit_distribution_temperature_low"
   IOField "I/O field_17" at 563,120 size 95x35; FormatPattern 9999
      ProcessValue <- "alarm_limit_preaheating_tank_pressure_low_delay"
   IOField "I/O field_18" at 563,160 size 95x35; FormatPattern 9999
      ProcessValue <- "alarm_limit_distribution_pressure_low_delay"
   IOField "I/O field_19" at 563,200 size 95x35; FormatPattern 9999
      ProcessValue <- "alarm_limit_preheating_temperature_low_delay"
   IOField "I/O field_20" at 563,240 size 95x35; FormatPattern 9999
      ProcessValue <- "alarm_limit_distribution_temperature_low_delay"
   Circle "Circle_7" at 671,120 size 30x30
      Appearance <- "preaheating_tank_pressure_low"
   IOField "I/O field_21" at 714,80 size 80x35; FormatPattern 999.9
      ProcessValue <- "sensor_inputs_preheating_steam_preassure"
   IOField "I/O field_22" at 714,120 size 80x35; FormatPattern 999.9
      ProcessValue <- "sensor_inputs_preheating_tank_pressure"
   IOField "I/O field_23" at 714,160 size 80x35; FormatPattern 999.9
      ProcessValue <- "sensor_inputs_distribution_tank_pressure"
   IOField "I/O field_24" at 714,200 size 80x35; FormatPattern 999.9
      ProcessValue <- "sensor_inputs_preheating_temperature"
   IOField "I/O field_25" at 714,240 size 80x35; FormatPattern 999.9
      ProcessValue <- "sensor_inputs_distribution_temperature"
   TextField "Text field_1" at 3,125 size 182x21; Text 'Heating Tank Pressure'
   TextField "Text field_2" at 3,166 size 213x21; Text 'Distribution Tank Pressure'
   TextField "Text field_3" at 3,208 size 215x21; Text 'Heating Tank Temperature'
   TextField "Text field_4" at 1,247 size 246x21; Text 'Distribution Tank Temperature'
   Circle "Circle_3" at 423,160 size 30x30
      Appearance <- "distribution_pressure_high"
   Circle "Circle_4" at 423,200 size 30x30
      Appearance <- "preheating_temperature_high"
   Circle "Circle_5" at 423,240 size 30x30
      Appearance <- "distribution_temperature_high"
   Circle "Circle_8" at 671,160 size 30x30
      Appearance <- "distribution_pressure_low"
   Circle "Circle_9" at 671,200 size 30x30
      Appearance <- "preheating_temperature_low"
   Circle "Circle_10" at 671,240 size 30x30
      Appearance <- "distribution_temperature_low"

screen "Alarm" 800x480, template "Lower Button"
   AlarmView "Alarm view_1" at 0,24 size 800x416

screen "System_Setpoints" 800x480, template "Lower Button"
   Button "Button_3" at 642,94 size 124x203; TextOff 'Text'
   Button "Button_15" at 29,259 size 230x36; TextOff 'Text'
   Button "Button_14" at 29,218 size 230x36; TextOff 'Text'
   Button "Button_13" at 29,177 size 230x36; TextOff 'Text'
   Button "Button_12" at 29,136 size 230x36; TextOff 'Text'
   Button "Button_11" at 29,95 size 230x36; TextOff 'Text'
   Button "Button_2" at 262,65 size 120x25; TextOff 'Setpoint'
   Button "Button_4" at 384,65 size 120x25; TextOff 'Tolerance'
   Button "Button_7" at 507,65 size 120x25; TextOff 'Process Value'
   Button "Button_8" at 262,94 size 367x203; TextOff 'Text'
   IOField "I/O field_5" at 267,96 size 115x35; FormatPattern 999.9
      ProcessValue <- "setpoint_preheating_steam_pressure"
   TextField "Text field_16" at 31,100 size 127x21; Text 'Steam Pressure'
   IOField "I/O field_1" at 388,96 size 115x35; FormatPattern 999.9
      ProcessValue <- "setpoint_preheating_steam_pressure_tolerance"
   IOField "I/O field_2" at 267,136 size 115x35; FormatPattern 999.9
      ProcessValue <- "setpoint_preheating_tank_pressure"
   IOField "I/O field_3" at 267,176 size 115x35; FormatPattern 999.9
      ProcessValue <- "setpoint_distribution_tank_pressure"
   IOField "I/O field_4" at 267,216 size 115x35; FormatPattern 999.9
      ProcessValue <- "setpoint_preheating_temperature"
   IOField "I/O field_6" at 267,256 size 115x35; FormatPattern 999.9
      ProcessValue <- "setpoint_distribution_temperature"
   IOField "I/O field_7" at 388,136 size 115x35; FormatPattern 999.9
      ProcessValue <- "setpoint_preaheating_tank_pressure_tolerance"
   IOField "I/O field_8" at 388,176 size 115x35; FormatPattern 999.9
      ProcessValue <- "setpoint_distribution_tank_pressure_tolerance"
   IOField "I/O field_9" at 388,216 size 115x35; FormatPattern 999.9
      ProcessValue <- "setpoint_preheating_temperature_tolerance"
   IOField "I/O field_10" at 388,256 size 115x35; FormatPattern 999.9
      ProcessValue <- "setpoint_distribution_temperature_tolerance"
   IOField "I/O field_21" at 510,96 size 115x35; FormatPattern 999.9
      ProcessValue <- "sensor_inputs_preheating_steam_preassure"
   IOField "I/O field_22" at 510,136 size 115x35; FormatPattern 999.9
      ProcessValue <- "sensor_inputs_preheating_tank_pressure"
   IOField "I/O field_23" at 510,176 size 115x35; FormatPattern 999.9
      ProcessValue <- "sensor_inputs_distribution_tank_pressure"
   IOField "I/O field_24" at 510,216 size 115x35; FormatPattern 999.9
      ProcessValue <- "sensor_inputs_preheating_temperature"
   IOField "I/O field_25" at 510,256 size 115x35; FormatPattern 999.9
      ProcessValue <- "sensor_inputs_distribution_temperature"
   TextField "Text field_1" at 30,141 size 182x21; Text 'Heating Tank Pressure'
   TextField "Text field_2" at 30,182 size 213x21; Text 'Distribution Tank Pressure'
   TextField "Text field_3" at 30,224 size 215x21; Text 'Heating Tank Temperature'
   TextField "Text field_4" at 29,264 size 246x21; Text 'Distribution Tank Temperature'
   Button "Button_1" at 645,65 size 120x25; TextOff 'Calibration'
   IOField "I/O field_11" at 647,96 size 115x35; FormatPattern 999.9
      ProcessValue <- "read_sensors_DB_Steam_pressure_input_Calibration"
   IOField "I/O field_12" at 647,136 size 115x35; FormatPattern 999.9
      ProcessValue <- "read_sensors_DB_preheating_tank_pressure_input_Calibration"
   IOField "I/O field_13" at 647,176 size 115x35; FormatPattern 999.9
      ProcessValue <- "read_sensors_DB_distribution_tank_pressure_input_Calibration"
   IOField "I/O field_14" at 647,216 size 115x35; FormatPattern 999.9
      ProcessValue <- "read_sensors_DB_preheating_temperature_input_Calibration"
   IOField "I/O field_15" at 647,256 size 115x35; FormatPattern 999.9
      ProcessValue <- "read_sensors_DB_distribution_temperature_input_Calibration"
   Button "Button_5" at 285,341 size 230x40; TextOff 'Preheating Tank PID Tuning'
      on Release: ActivateScreen("PT_PID_Tuning", 0)
   Button "Button_6" at 285,384 size 230x40; TextOff 'Distribution Tank PID Tuning'
      on Release: ActivateScreen("DT_PID_Tuning", 0)

screen "Trend" 800x480, template "Lower Button"
   TrendView "Trend view_1" at 6,40 size 786x382
   Button "Button_10" at 240,7 size 320x28; TextOff 'Distribution Tank Temperature'

PopupScreen "V-PV" 185x95
   GraphicView "V-D Off" at 126,6 size 45x35; Picture "Graphic_37"
      Visibility <- "preheating_vent"
   GraphicView "V-D On" at 126,6 size 45x35; Picture "Graphic_38"
      Visibility <- "preheating_vent"
   Button "Button_1" at 2,3 size 180x40; TextOff 'Preheating Vent Valve'
   Button "Button_5" at 2,42 size 180x50; TextOff 'Manual Operation'
   Button "Button_6" at 5,57 size 85x32; TextOff 'Start'
      on Press: SetBit("manual_preheating_vent")
   Button "Button_7" at 94,57 size 85x32; TextOff 'Stop'
      on Press: ResetBit("manual_preheating_vent")
   Group "V-D" at 126,6 size 45x35; Picture "Graphic_37"

PopupScreen "V-DV" 185x95
   GraphicView "V-D Off" at 126,6 size 45x35; Picture "Graphic_37"
      Visibility <- "distribution_vent"
   GraphicView "V-D On" at 126,6 size 45x35; Picture "Graphic_38"
      Visibility <- "distribution_vent"
   Button "Button_1" at 2,3 size 180x40; TextOff 'Distribution Vent Valve'
   Button "Button_5" at 2,42 size 180x50; TextOff 'Manual Operation'
   Button "Button_6" at 5,57 size 85x32; TextOff 'Start'
      on Press: ResetBit("manual_distribution_vent")
   Button "Button_7" at 94,57 size 85x32; TextOff 'Stop'
      on Press: SetBit("manual_distribution_vent")
   Group "V-D" at 126,6 size 45x35; Picture "Graphic_37"

screen "DT_PID_Tuning" 800x480, template "Lower Button"
   Button "Button_10" at 344,10 size 261x50; TextOff 'Distribution Tank'
   Button "Button_15" at 98,224 size 240x36; TextOff 'Text'
   Button "Button_14" at 98,184 size 240x35; TextOff 'Text'
   Button "Button_13" at 98,144 size 240x35; TextOff 'Text'
   Button "Button_12" at 98,104 size 240x35; TextOff 'Text'
   Button "Button_11" at 98,64 size 240x35; TextOff 'Text'
   Button "Button_2" at 346,33 size 125x25; TextOff 'Heat'
   Button "Button_4" at 478,33 size 125x25; TextOff 'Cool'
   Button "Button_8" at 343,62 size 264x360; TextOff 'Text'
   IOField "I/O field_5" at 346,64 size 125x35; FormatPattern 999.9
      ProcessValue <- "Gain"
   TextField "Text field_16" at 100,70 size 142x21; Text 'Proportional Gain'
   IOField "I/O field_2" at 346,104 size 125x35; FormatPattern 999.9
      ProcessValue <- "Ti"
   IOField "I/O field_3" at 346,144 size 125x35; FormatPattern 999.9
      ProcessValue <- "Td"
   IOField "I/O field_4" at 346,184 size 125x35; FormatPattern 999.9
      ProcessValue <- "TdFiltRatio"
   IOField "I/O field_6" at 346,224 size 125x35; FormatPattern 999.9
      ProcessValue <- "PWeighting"
   TextField "Text field_1" at 99,109 size 193x21; Text 'Integral Action Time (s)'
   TextField "Text field_2" at 99,150 size 207x21; Text 'Derivative Action Time (s)'
   TextField "Text field_3" at 99,192 size 215x21; Text 'Derivative delay coefficient'
   TextField "Text field_4" at 98,232 size 232x21; Text 'Proportinal Action Weighting'
   Button "Button_3" at 98,264 size 240x36; TextOff 'Text'
   TextField "Text field_5" at 98,272 size 222x21; Text 'Derivative Action Weighting'
   Button "Button_5" at 98,304 size 240x36; TextOff 'Text'
   TextField "Text field_6" at 98,312 size 170x21; Text 'Sampling time of PID'
   Button "Button_6" at 98,344 size 240x36; TextOff 'Text'
   TextField "Text field_7" at 98,352 size 135x21; Text 'Dead zone width'
   Button "Button_9" at 98,384 size 240x36; TextOff 'Text'
   TextField "Text field_8" at 98,392 size 155x21; Text 'Control zone width'
   IOField "I/O field_11" at 346,264 size 125x35; FormatPattern 999.9
      ProcessValue <- "DWeighting"
   IOField "I/O field_12" at 346,304 size 125x35; FormatPattern 999.9
      ProcessValue <- "Cycle"
   IOField "I/O field_13" at 346,344 size 125x35; FormatPattern 999.9
      ProcessValue <- "DeadZone"
   IOField "I/O field_14" at 346,384 size 125x35; FormatPattern 999.9
      ProcessValue <- "ControlZone"
   IOField "I/O field_1" at 477,64 size 125x35; FormatPattern 999.9
      ProcessValue <- "Gain"
   IOField "I/O field_7" at 477,104 size 125x35; FormatPattern 999.9
      ProcessValue <- "Ti"
   IOField "I/O field_8" at 477,144 size 125x35; FormatPattern 999.9
      ProcessValue <- "Td"
   IOField "I/O field_9" at 477,184 size 125x35; FormatPattern 999.9
      ProcessValue <- "TdFiltRatio"
   IOField "I/O field_10" at 477,224 size 125x35; FormatPattern 999.9
      ProcessValue <- "PWeighting"
   IOField "I/O field_15" at 477,264 size 125x35; FormatPattern 999.9
      ProcessValue <- "DWeighting"
   IOField "I/O field_16" at 477,304 size 125x35; FormatPattern 999.9
      ProcessValue <- "Cycle"
   IOField "I/O field_17" at 477,344 size 125x35; FormatPattern 999.9
      ProcessValue <- "DeadZone"
   IOField "I/O field_18" at 477,384 size 125x35; FormatPattern 999.9
      ProcessValue <- "ControlZone"
   Button "Button_1" at 640,397 size 160x40; TextOff 'Trend'
      on Release: ActivateScreen("DT_Trend", 0)

screen "DT_Trend" 800x480, template "Lower Button"
   TrendView "Trend view_1" at 5,37 size 789x358
   Button "Button_4" at 0,397 size 160x40; TextOff 'Previous'
      on Release: ActivateScreen("DT_PID_Tuning", 0)
   Button "Button_10" at 240,7 size 320x28; TextOff 'Distribution Tank Temperature Trend'
   TextField "Text field_1" at 658,364 size 28x23; Text 'SP'
   TextField "Text field_2" at 714,364 size 29x23; Text 'PV'

screen "PT_PID_Tuning" 800x480, template "Lower Button"
   Button "Button_10" at 344,10 size 261x50; TextOff 'Preheating Tank'
   Button "Button_15" at 98,224 size 240x36; TextOff 'Text'
   Button "Button_14" at 98,184 size 240x35; TextOff 'Text'
   Button "Button_13" at 98,144 size 240x35; TextOff 'Text'
   Button "Button_12" at 98,104 size 240x35; TextOff 'Text'
   Button "Button_11" at 98,64 size 240x35; TextOff 'Text'
   Button "Button_2" at 346,33 size 125x25; TextOff 'Heat'
   Button "Button_4" at 478,33 size 125x25; TextOff 'Cool'
   Button "Button_8" at 343,62 size 264x360; TextOff 'Text'
   IOField "I/O field_5" at 346,64 size 125x35; FormatPattern 999.9
      ProcessValue <- "Gain"
   TextField "Text field_16" at 100,70 size 142x21; Text 'Proportional Gain'
   IOField "I/O field_2" at 346,104 size 125x35; FormatPattern 999.9
      ProcessValue <- "Ti"
   IOField "I/O field_3" at 346,144 size 125x35; FormatPattern 999.9
      ProcessValue <- "Td"
   IOField "I/O field_4" at 346,184 size 125x35; FormatPattern 999.9
      ProcessValue <- "TdFiltRatio"
   IOField "I/O field_6" at 346,224 size 125x35; FormatPattern 999.9
      ProcessValue <- "PWeighting"
   TextField "Text field_1" at 99,109 size 193x21; Text 'Integral Action Time (s)'
   TextField "Text field_2" at 99,150 size 207x21; Text 'Derivative Action Time (s)'
   TextField "Text field_3" at 99,192 size 215x21; Text 'Derivative delay coefficient'
   TextField "Text field_4" at 98,232 size 232x21; Text 'Proportinal Action Weighting'
   Button "Button_3" at 98,264 size 240x36; TextOff 'Text'
   TextField "Text field_5" at 98,272 size 222x21; Text 'Derivative Action Weighting'
   Button "Button_5" at 98,304 size 240x36; TextOff 'Text'
   TextField "Text field_6" at 98,312 size 170x21; Text 'Sampling time of PID'
   Button "Button_6" at 98,344 size 240x36; TextOff 'Text'
   TextField "Text field_7" at 98,352 size 135x21; Text 'Dead zone width'
   Button "Button_9" at 98,384 size 240x36; TextOff 'Text'
   TextField "Text field_8" at 98,392 size 155x21; Text 'Control zone width'
   IOField "I/O field_11" at 346,264 size 125x35; FormatPattern 999.9
      ProcessValue <- "DWeighting"
   IOField "I/O field_12" at 346,304 size 125x35; FormatPattern 999.9
      ProcessValue <- "Cycle"
   IOField "I/O field_13" at 346,344 size 125x35; FormatPattern 999.9
      ProcessValue <- "DeadZone"
   IOField "I/O field_14" at 346,384 size 125x35; FormatPattern 999.9
      ProcessValue <- "ControlZone"
   IOField "I/O field_1" at 477,64 size 125x35; FormatPattern 999.9
      ProcessValue <- "Gain"
   IOField "I/O field_7" at 477,104 size 125x35; FormatPattern 999.9
      ProcessValue <- "Ti"
   IOField "I/O field_8" at 477,144 size 125x35; FormatPattern 999.9
      ProcessValue <- "Td"
   IOField "I/O field_9" at 477,184 size 125x35; FormatPattern 999.9
      ProcessValue <- "TdFiltRatio"
   IOField "I/O field_10" at 477,224 size 125x35; FormatPattern 999.9
      ProcessValue <- "PWeighting"
   IOField "I/O field_15" at 477,264 size 125x35; FormatPattern 999.9
      ProcessValue <- "DWeighting"
   IOField "I/O field_16" at 477,304 size 125x35; FormatPattern 999.9
      ProcessValue <- "Cycle"
   IOField "I/O field_17" at 477,344 size 125x35; FormatPattern 999.9
      ProcessValue <- "DeadZone"
   IOField "I/O field_18" at 477,384 size 125x35; FormatPattern 999.9
      ProcessValue <- "ControlZone"
   Button "Button_1" at 640,397 size 160x40; TextOff 'Trend'
      on Release: ActivateScreen("PT_Trend", 0)

screen "PT_Trend" 800x480, template "Lower Button"
   TrendView "Trend view_1" at 5,37 size 789x358
   Button "Button_4" at 0,397 size 160x40; TextOff 'Previous'
      on Release: ActivateScreen("PT_PID_Tuning", 0)
   Button "Button_10" at 240,7 size 320x28; TextOff 'Preheating Tank Temperature Trend'
   TextField "Text field_1" at 658,364 size 28x23; Text 'SP'
   TextField "Text field_2" at 714,364 size 29x23; Text 'PV'
*)